LIN {X 0,Y 355.726,Z 424.465,A -85,B 0,C 180,E1 -13380.407,E2 -13380.407} C_VEL
LIN {X 0,Y 354.984,Z 431.448,A -85,B 0,C 180,E1 -13384.185,E2 -13384.185} C_VEL
LIN {X 0,Y 354.319,Z 439.711,A -85,B 0,C 180,E1 -13388.41,E2 -13388.41} C_VEL
LIN {X 0,Y 357.709,Z 454.995,A -85,B 0,C 180,E1 -13389.372,E2 -13389.372} C_VEL
LIN {X 0,Y 359.439,Z 467.166,A -85,B 0,C 180,E1 -13390.263,E2 -13390.263} C_VEL
LIN {X 0,Y 360.148,Z 480.167,A -85,B 0,C 180,E1 -13391.37,E2 -13391.37} C_VEL
LIN {X 0,Y 359.701,Z 487.628,A -85,B 0,C 180,E1 -13392.082,E2 -13392.082} C_VEL
LIN {X 0,Y 358.234,Z 498.948,A -85,B 0,C 180,E1 -13393.331,E2 -13393.331} C_VEL
LIN {X 0,Y 356.998,Z 508.224,A -85,B 0,C 180,E1 -13394.593,E2 -13394.593} C_VEL
LIN {X 0,Y 356.085,Z 516.778,A -85,B 0,C 180,E1 -13396.013,E2 -13396.013} C_VEL
LIN {X 0,Y 355.032,Z 525.202,A -85,B 0,C 180,E1 -13397.718,E2 -13397.718} C_VEL
LIN {X 0,Y 354.24,Z 532.058,A -85,B 0,C 180,E1 -13399.43,E2 -13399.43} C_VEL
LIN {X 0,Y 353.672,Z 538.425,A -85,B 0,C 180,E1 -13401.433,E2 -13401.433} C_VEL
LIN {X 0,Y 353.414,Z 542.602,A -85,B 0,C 180,E1 -13403.152,E2 -13403.152} C_VEL
LIN {X 0,Y 353.311,Z 544.771,A -85,B 0,C 180,E1 -13404.296,E2 -13404.296} C_VEL
LIN {X 0,Y 353.316,Z 546.521,A -85,B 0,C 180,E1 -13405.441,E2 -13405.441} C_VEL
LIN {X 0,Y 353.284,Z 547.858,A -85,B 0,C 180,E1 -13406.583,E2 -13406.583} C_VEL
LIN {X 0,Y 353.35,Z 548.753,A -85,B 0,C 180,E1 -13407.724,E2 -13407.724} C_VEL
LIN {X 0,Y 353.463,Z 549.226,A -85,B 0,C 180,E1 -13408.865,E2 -13408.865} C_VEL
LIN {X 0,Y 353.456,Z 549.291,A -85,B 0,C 180,E1 -13410.004,E2 -13410.004} C_VEL
LIN {X 0,Y 353.47,Z 548.959,A -85,B 0,C 180,E1 -13411.143,E2 -13411.143} C_VEL
LIN {X 0,Y 353.41,Z 548.175,A -85,B 0,C 180,E1 -13412.284,E2 -13412.284} C_VEL
LIN {X 0,Y 353.313,Z 546.954,A -85,B 0,C 180,E1 -13413.425,E2 -13413.425} C_VEL
LIN {X 0,Y 353.368,Z 544.327,A -85,B 0,C 180,E1 -13415.139,E2 -13415.139} C_VEL
LIN {X 0,Y 353.432,Z 540.637,A -85,B 0,C 180,E1 -13416.856,E2 -13416.856} C_VEL
LIN {X 0,Y 353.674,Z 535.798,A -85,B 0,C 180,E1 -13418.575,E2 -13418.575} C_VEL
LIN {X 0,Y 354.06,Z 529.666,A -85,B 0,C 180,E1 -13420.295,E2 -13420.295} C_VEL
LIN {X 0,Y 354.749,Z 522.044,A -85,B 0,C 180,E1 -13422.01,E2 -13422.01} C_VEL
LIN {X 0,Y 355.442,Z 514.243,A -85,B 0,C 180,E1 -13423.438,E2 -13423.438} C_VEL
LIN {X 0,Y 356.383,Z 503.675,A -85,B 0,C 180,E1 -13425.004,E2 -13425.004} C_VEL
LIN {X 0,Y 357.344,Z 493,A -85,B 0,C 180,E1 -13426.279,E2 -13426.279} C_VEL
LIN {X 0,Y 358.499,Z 481.057,A -85,B 0,C 180,E1 -13427.399,E2 -13427.399} C_VEL
LIN {X 0,Y 357.508,Z 469.159,A -85,B 0,C 180,E1 -13428.336,E2 -13428.336} C_VEL
LIN {X 0,Y 355.884,Z 455.898,A -85,B 0,C 180,E1 -13429.157,E2 -13429.157} C_VEL
LIN {X 0,Y 354,Z 442.82,A -85,B 0,C 180,E1 -13429.766,E2 -13429.766} C_VEL
LIN {X 0,Y 354.506,Z 435.528,A -85,B 0,C 180,E1 -13433.363,E2 -13433.363} C_VEL
LIN {X 0,Y 355.125,Z 428.123,A -85,B 0,C 180,E1 -13437.08,E2 -13437.08} C_VEL
LIN {X 0,Y 355.948,Z 420.705,A -85,B 0,C 180,E1 -13440.891,E2 -13440.891} C_VEL
LIN {X 0,Y 356.669,Z 414.53,A -85,B 0,C 180,E1 -13444.147,E2 -13444.147} C_VEL
LIN {X 0,Y 357.086,Z 410.748,A -85,B 0,C 180,E1 -13446.2,E2 -13446.2} C_VEL
LIN {X 0,Y 356.797,Z 407.568,A -85,B 0,C 180,E1 -13448.009,E2 -13448.009} C_VEL
LIN {X 0,Y 355.865,Z 401.962,A -85,B 0,C 180,E1 -13451.368,E2 -13451.368} C_VEL
LIN {X 0,Y 354.819,Z 396.286,A -85,B 0,C 180,E1 -13454.988,E2 -13454.988} C_VEL
LIN {X 0,Y 354.786,Z 396.293,A -85,B 0,C 180,E1 -13458.833,E2 -13458.833} C_VEL
LIN {X 0,Y 354.814,Z 396.285,A -85,B 0,C 180,E1 -13462.406,E2 -13462.406} C_VEL
LIN {X 0,Y 354.823,Z 396.288,A -85,B 0,C 180,E1 -13464.941,E2 -13464.941} C_VEL
LIN {X 0,Y 354.808,Z 396.287,A -85,B 0,C 180,E1 -13468.406,E2 -13468.406} C_VEL
LIN {X 0,Y 354.817,Z 396.287,A -85,B 0,C 180,E1 -13471.615,E2 -13471.615} C_VEL
LIN {X 0,Y 354.85,Z 396.282,A -85,B 0,C 180,E1 -13475.657,E2 -13475.657} C_VEL
LIN {X 0,Y 354.841,Z 396.287,A -85,B 0,C 180,E1 -13479.113,E2 -13479.113} C_VEL
LIN {X 0,Y 354.895,Z 396.278,A -85,B 0,C 180,E1 -13482.719,E2 -13482.719} C_VEL
LIN {X 0,Y 354.966,Z 396.266,A -85,B 0,C 180,E1 -13486.255,E2 -13486.255} C_VEL
LIN {X 0,Y 354.969,Z 396.266,A -85,B 0,C 180,E1 -13489.735,E2 -13489.735} C_VEL
LIN {X 0,Y 355.12,Z 396.251,A -85,B 0,C 180,E1 -13493.179,E2 -13493.179} C_VEL
LIN {X 0,Y 355.254,Z 396.231,A -85,B 0,C 180,E1 -13497.731,E2 -13497.731} C_VEL
LIN {X 0,Y 355.345,Z 396.219,A -85,B 0,C 180,E1 -13499.999,E2 -13499.999} C_VEL
LIN {X 0,Y 355.246,Z 396.233,A -85,B 0,C 180,E1 -13502.267,E2 -13502.267} C_VEL
LIN {X 0,Y 355.1,Z 396.255,A -85,B 0,C 180,E1 -13506.819,E2 -13506.819} C_VEL
LIN {X 0,Y 354.967,Z 396.268,A -85,B 0,C 180,E1 -13510.263,E2 -13510.263} C_VEL
LIN {X 0,Y 354.955,Z 396.268,A -85,B 0,C 180,E1 -13514.017,E2 -13514.017} C_VEL
LIN {X 0,Y 354.902,Z 396.275,A -85,B 0,C 180,E1 -13518.09,E2 -13518.09} C_VEL
LIN {X 0,Y 354.826,Z 396.285,A -85,B 0,C 180,E1 -13522.105,E2 -13522.105} C_VEL
LIN {X 0,Y 354.908,Z 396.274,A -85,B 0,C 180,E1 -13525.825,E2 -13525.825} C_VEL
LIN {X 0,Y 354.815,Z 396.285,A -85,B 0,C 180,E1 -13529.681,E2 -13529.681} C_VEL
LIN {X 0,Y 354.824,Z 396.284,A -85,B 0,C 180,E1 -13533.681,E2 -13533.681} C_VEL
LIN {X 0,Y 354.805,Z 396.291,A -85,B 0,C 180,E1 -13536.457,E2 -13536.457} C_VEL
LIN {X 0,Y 354.807,Z 396.286,A -85,B 0,C 180,E1 -13539.416,E2 -13539.416} C_VEL
LIN {X 0,Y 354.794,Z 396.291,A -85,B 0,C 180,E1 -13542.864,E2 -13542.864} C_VEL
LIN {X 0,Y 354.772,Z 396.293,A -85,B 0,C 180,E1 -13546.1,E2 -13546.1} C_VEL
LIN {X 0,Y 354.79,Z 396.289,A -85,B 0,C 180,E1 -13549.175,E2 -13549.175} C_VEL
LIN {X 0,Y 354.81,Z 396.291,A -85,B 0,C 180,E1 -13552.4,E2 -13552.4} C_VEL
LIN {X 0,Y 354.816,Z 396.287,A -85,B 0,C 180,E1 -13554.937,E2 -13554.937} C_VEL
LIN {X 0,Y 354.797,Z 396.292,A -85,B 0,C 180,E1 -13558.402,E2 -13558.402} C_VEL
LIN {X 0,Y 354.849,Z 396.281,A -85,B 0,C 180,E1 -13561.615,E2 -13561.615} C_VEL
LIN {X 0,Y 354.901,Z 396.279,A -85,B 0,C 180,E1 -13564.169,E2 -13564.169} C_VEL
LIN {X 0,Y 354.836,Z 396.285,A -85,B 0,C 180,E1 -13567.89,E2 -13567.89} C_VEL
LIN {X 0,Y 354.922,Z 396.274,A -85,B 0,C 180,E1 -13571.888,E2 -13571.888} C_VEL
LIN {X 0,Y 354.941,Z 396.273,A -85,B 0,C 180,E1 -13575.977,E2 -13575.977} C_VEL
LIN {X 0,Y 354.975,Z 396.267,A -85,B 0,C 180,E1 -13579.732,E2 -13579.732} C_VEL
LIN {X 0,Y 355.12,Z 396.247,A -85,B 0,C 180,E1 -13583.176,E2 -13583.176} C_VEL
LIN {X 0,Y 355.237,Z 396.235,A -85,B 0,C 180,E1 -13587.728,E2 -13587.728} C_VEL
LIN {X 0,Y 355.388,Z 396.218,A -85,B 0,C 180,E1 -13589.996,E2 -13589.996} C_VEL
LIN {X 0,Y 355.237,Z 396.238,A -85,B 0,C 180,E1 -13592.263,E2 -13592.263} C_VEL
LIN {X 0,Y 355.128,Z 396.247,A -85,B 0,C 180,E1 -13596.815,E2 -13596.815} C_VEL
LIN {X 0,Y 355.005,Z 396.262,A -85,B 0,C 180,E1 -13599.108,E2 -13599.108} C_VEL
LIN {X 0,Y 354.913,Z 396.275,A -85,B 0,C 180,E1 -13602.576,E2 -13602.576} C_VEL
LIN {X 0,Y 354.877,Z 396.283,A -85,B 0,C 180,E1 -13606.092,E2 -13606.092} C_VEL
LIN {X 0,Y 354.89,Z 396.278,A -85,B 0,C 180,E1 -13608.468,E2 -13608.468} C_VEL
LIN {X 0,Y 354.816,Z 396.29,A -85,B 0,C 180,E1 -13612.102,E2 -13612.102} C_VEL
LIN {X 0,Y 354.828,Z 396.284,A -85,B 0,C 180,E1 -13614.573,E2 -13614.573} C_VEL
LIN {X 0,Y 354.671,Z 396.303,A -85,B 0,C 180,E1 -13617.108,E2 -13617.108} C_VEL
LIN {X 0,Y 354.374,Z 396.345,A -85,B 0,C 180,E1 -13619.717,E2 -13619.717} C_VEL
LIN {X 0,Y 354.027,Z 396.387,A -85,B 0,C 180,E1 -13622.405,E2 -13622.405} C_VEL
LIN {X 0,Y 353.895,Z 396.822,A -85,B 0,C 180,E1 -13623.777,E2 -13623.777} C_VEL
LIN {X 0,Y 353.774,Z 400.146,A -85,B 0,C 180,E1 -13627.382,E2 -13627.382} C_VEL
LIN {X 0,Y 353.684,Z 403.57,A -85,B 0,C 180,E1 -13630.969,E2 -13630.969} C_VEL
LIN {X 0,Y 353.68,Z 404.977,A -85,B 0,C 180,E1 -13632.398,E2 -13632.398} C_VEL
LIN {X 0,Y 356.886,Z 418.397,A -85,B 0,C 180,E1 -13633.129,E2 -13633.129} C_VEL
LIN {X 0,Y 359.642,Z 431.249,A -85,B 0,C 180,E1 -13634.039,E2 -13634.039} C_VEL
LIN {X 0,Y 359.648,Z 436.037,A -85,B 0,C 180,E1 -13634.399,E2 -13634.399} C_VEL
LIN {X 0,Y 358.833,Z 447.243,A -85,B 0,C 180,E1 -13635.363,E2 -13635.363} C_VEL
LIN {X 0,Y 357.756,Z 458.778,A -85,B 0,C 180,E1 -13636.615,E2 -13636.615} C_VEL
LIN {X 0,Y 357.607,Z 460.555,A -85,B 0,C 180,E1 -13636.835,E2 -13636.835} C_VEL
LIN {X 0,Y 356.539,Z 465.133,A -85,B 0,C 180,E1 -13637.412,E2 -13637.412} C_VEL
LIN {X 0,Y 353.076,Z 472.268,A -85,B 0,C 180,E1 -13638.376,E2 -13638.376} C_VEL
LIN {X 0,Y 349.606,Z 478.873,A -85,B 0,C 180,E1 -13639.445,E2 -13639.445} C_VEL
LIN {X 0,Y 348.543,Z 482.621,A -85,B 0,C 180,E1 -13640.176,E2 -13640.176} C_VEL
LIN {X 0,Y 347.827,Z 490.364,A -85,B 0,C 180,E1 -13641.991,E2 -13641.991} C_VEL
LIN {X 0,Y 347.238,Z 496.207,A -85,B 0,C 180,E1 -13643.702,E2 -13643.702} C_VEL
LIN {X 0,Y 346.846,Z 500.886,A -85,B 0,C 180,E1 -13645.436,E2 -13645.436} C_VEL
LIN {X 0,Y 346.507,Z 504.996,A -85,B 0,C 180,E1 -13647.489,E2 -13647.489} C_VEL
LIN {X 0,Y 346.224,Z 507.705,A -85,B 0,C 180,E1 -13649.506,E2 -13649.506} C_VEL
LIN {X 0,Y 346.209,Z 508.83,A -85,B 0,C 180,E1 -13650.845,E2 -13650.845} C_VEL
LIN {X 0,Y 346.169,Z 509.366,A -85,B 0,C 180,E1 -13652.165,E2 -13652.165} C_VEL
LIN {X 0,Y 346.207,Z 509.422,A -85,B 0,C 180,E1 -13653.476,E2 -13653.476} C_VEL
LIN {X 0,Y 346.334,Z 508.95,A -85,B 0,C 180,E1 -13654.778,E2 -13654.778} C_VEL
LIN {X 0,Y 346.526,Z 507.981,A -85,B 0,C 180,E1 -13656.071,E2 -13656.071} C_VEL
LIN {X 0,Y 346.814,Z 506.542,A -85,B 0,C 180,E1 -13657.356,E2 -13657.356} C_VEL
LIN {X 0,Y 347.305,Z 503.406,A -85,B 0,C 180,E1 -13659.261,E2 -13659.261} C_VEL
LIN {X 0,Y 347.906,Z 499.097,A -85,B 0,C 180,E1 -13661.144,E2 -13661.144} C_VEL
LIN {X 0,Y 348.766,Z 493.475,A -85,B 0,C 180,E1 -13663.012,E2 -13663.012} C_VEL
LIN {X 0,Y 349.903,Z 486.366,A -85,B 0,C 180,E1 -13664.865,E2 -13664.865} C_VEL
LIN {X 0,Y 351.209,Z 477.432,A -85,B 0,C 180,E1 -13666.697,E2 -13666.697} C_VEL
LIN {X 0,Y 352.565,Z 467.814,A -85,B 0,C 180,E1 -13668.283,E2 -13668.283} C_VEL
LIN {X 0,Y 353.916,Z 458.132,A -85,B 0,C 180,E1 -13669.561,E2 -13669.561} C_VEL
LIN {X 0,Y 355.189,Z 447.027,A -85,B 0,C 180,E1 -13670.75,E2 -13670.75} C_VEL
LIN {X 0,Y 356.058,Z 438.589,A -85,B 0,C 180,E1 -13671.487,E2 -13671.487} C_VEL
LIN {X 0,Y 354.629,Z 430.955,A -85,B 0,C 180,E1 -13672.218,E2 -13672.218} C_VEL
LIN {X 0,Y 351.014,Z 418.776,A -85,B 0,C 180,E1 -13673.318,E2 -13673.318} C_VEL
LIN {X 0,Y 347.558,Z 409.355,A -85,B 0,C 180,E1 -13674.089,E2 -13674.089} C_VEL
LIN {X 0,Y 347.468,Z 408.819,A -85,B 0,C 180,E1 -13674.124,E2 -13674.124} C_VEL
LIN {X 0,Y 347.648,Z 405.401,A -85,B 0,C 180,E1 -13678.843,E2 -13678.843} C_VEL
LIN {X 0,Y 348.104,Z 403.772,A -85,B 0,C 180,E1 -13681.158,E2 -13681.158} C_VEL
LIN {X 0,Y 348.199,Z 400.872,A -85,B 0,C 180,E1 -13685.793,E2 -13685.793} C_VEL
LIN {X 0,Y 348.303,Z 399.27,A -85,B 0,C 180,E1 -13688.656,E2 -13688.656} C_VEL
LIN {X 0,Y 347.865,Z 397.31,A -85,B 0,C 180,E1 -13692.841,E2 -13692.841} C_VEL
LIN {X 0,Y 347.839,Z 397.157,A -85,B 0,C 180,E1 -13695.229,E2 -13695.229} C_VEL
LIN {X 0,Y 347.833,Z 397.16,A -85,B 0,C 180,E1 -13698.862,E2 -13698.862} C_VEL
LIN {X 0,Y 347.781,Z 397.163,A -85,B 0,C 180,E1 -13702.58,E2 -13702.58} C_VEL
LIN {X 0,Y 347.792,Z 397.164,A -85,B 0,C 180,E1 -13705.111,E2 -13705.111} C_VEL
LIN {X 0,Y 347.783,Z 397.162,A -85,B 0,C 180,E1 -13707.697,E2 -13707.697} C_VEL
LIN {X 0,Y 347.736,Z 397.171,A -85,B 0,C 180,E1 -13710.35,E2 -13710.35} C_VEL
LIN {X 0,Y 347.718,Z 397.171,A -85,B 0,C 180,E1 -13714.468,E2 -13714.468} C_VEL
LIN {X 0,Y 347.746,Z 397.169,A -85,B 0,C 180,E1 -13716.069,E2 -13716.069} C_VEL
LIN {X 0,Y 348.261,Z 399.777,A -85,B 0,C 180,E1 -13720.224,E2 -13720.224} C_VEL
LIN {X 0,Y 348.756,Z 402.481,A -85,B 0,C 180,E1 -13723.501,E2 -13723.501} C_VEL
LIN {X 0,Y 349.311,Z 405.852,A -85,B 0,C 180,E1 -13726.845,E2 -13726.845} C_VEL
LIN {X 0,Y 349.963,Z 409.541,A -85,B 0,C 180,E1 -13730.019,E2 -13730.019} C_VEL
LIN {X 0,Y 350.447,Z 413.541,A -85,B 0,C 180,E1 -13733.02,E2 -13733.02} C_VEL
LIN {X 0,Y 350.372,Z 415.65,A -85,B 0,C 180,E1 -13734.436,E2 -13734.436} C_VEL
LIN {X 0,Y 349.443,Z 420.778,A -85,B 0,C 180,E1 -13737.642,E2 -13737.642} C_VEL
LIN {X 0,Y 348.397,Z 427.812,A -85,B 0,C 180,E1 -13741.708,E2 -13741.708} C_VEL
LIN {X 0,Y 347.786,Z 433.661,A -85,B 0,C 180,E1 -13744.895,E2 -13744.895} C_VEL
LIN {X 0,Y 347.336,Z 439.222,A -85,B 0,C 180,E1 -13747.806,E2 -13747.806} C_VEL
LIN {X 0,Y 350.654,Z 453.448,A -85,B 0,C 180,E1 -13748.749,E2 -13748.749} C_VEL
LIN {X 0,Y 352.665,Z 466.488,A -85,B 0,C 180,E1 -13749.735,E2 -13749.735} C_VEL
LIN {X 0,Y 353.413,Z 479.258,A -85,B 0,C 180,E1 -13750.85,E2 -13750.85} C_VEL
LIN {X 0,Y 353.155,Z 486.716,A -85,B 0,C 180,E1 -13751.589,E2 -13751.589} C_VEL
LIN {X 0,Y 351.618,Z 498.048,A -85,B 0,C 180,E1 -13752.858,E2 -13752.858} C_VEL
LIN {X 0,Y 350.161,Z 508.316,A -85,B 0,C 180,E1 -13754.284,E2 -13754.284} C_VEL
LIN {X 0,Y 349.163,Z 516.792,A -85,B 0,C 180,E1 -13755.735,E2 -13755.735} C_VEL
LIN {X 0,Y 348.076,Z 525.127,A -85,B 0,C 180,E1 -13757.469,E2 -13757.469} C_VEL
LIN {X 0,Y 347.205,Z 531.924,A -85,B 0,C 180,E1 -13759.213,E2 -13759.213} C_VEL
LIN {X 0,Y 346.63,Z 538.191,A -85,B 0,C 180,E1 -13761.258,E2 -13761.258} C_VEL
LIN {X 0,Y 346.339,Z 542.311,A -85,B 0,C 180,E1 -13763.011,E2 -13763.011} C_VEL
LIN {X 0,Y 346.23,Z 544.459,A -85,B 0,C 180,E1 -13764.179,E2 -13764.179} C_VEL
LIN {X 0,Y 346.228,Z 546.191,A -85,B 0,C 180,E1 -13765.347,E2 -13765.347} C_VEL
LIN {X 0,Y 346.204,Z 547.505,A -85,B 0,C 180,E1 -13766.513,E2 -13766.513} C_VEL
LIN {X 0,Y 346.252,Z 548.363,A -85,B 0,C 180,E1 -13767.678,E2 -13767.678} C_VEL
LIN {X 0,Y 346.379,Z 548.818,A -85,B 0,C 180,E1 -13768.842,E2 -13768.842} C_VEL
LIN {X 0,Y 346.393,Z 548.866,A -85,B 0,C 180,E1 -13770.004,E2 -13770.004} C_VEL
LIN {X 0,Y 346.406,Z 548.506,A -85,B 0,C 180,E1 -13771.167,E2 -13771.167} C_VEL
LIN {X 0,Y 346.314,Z 547.681,A -85,B 0,C 180,E1 -13772.33,E2 -13772.33} C_VEL
LIN {X 0,Y 346.235,Z 546.439,A -85,B 0,C 180,E1 -13773.495,E2 -13773.495} C_VEL
LIN {X 0,Y 346.291,Z 543.763,A -85,B 0,C 180,E1 -13775.244,E2 -13775.244} C_VEL
LIN {X 0,Y 346.376,Z 540.02,A -85,B 0,C 180,E1 -13776.997,E2 -13776.997} C_VEL
LIN {X 0,Y 346.621,Z 535.123,A -85,B 0,C 180,E1 -13778.751,E2 -13778.751} C_VEL
LIN {X 0,Y 346.997,Z 528.923,A -85,B 0,C 180,E1 -13780.507,E2 -13780.507} C_VEL
LIN {X 0,Y 347.743,Z 521.212,A -85,B 0,C 180,E1 -13782.256,E2 -13782.256} C_VEL
LIN {X 0,Y 348.699,Z 511.532,A -85,B 0,C 180,E1 -13784,E2 -13784} C_VEL
LIN {X 0,Y 349.491,Z 502.638,A -85,B 0,C 180,E1 -13785.307,E2 -13785.307} C_VEL
LIN {X 0,Y 350.474,Z 491.799,A -85,B 0,C 180,E1 -13786.608,E2 -13786.608} C_VEL
LIN {X 0,Y 351.5,Z 481.346,A -85,B 0,C 180,E1 -13787.606,E2 -13787.606} C_VEL
LIN {X 0,Y 350.414,Z 468.521,A -85,B 0,C 180,E1 -13788.645,E2 -13788.645} C_VEL
LIN {X 0,Y 348.819,Z 455.316,A -85,B 0,C 180,E1 -13789.478,E2 -13789.478} C_VEL
LIN {X 0,Y 346.964,Z 442.526,A -85,B 0,C 180,E1 -13790.068,E2 -13790.068} C_VEL
LIN {X 0,Y 347.512,Z 435.034,A -85,B 0,C 180,E1 -13793.862,E2 -13793.862} C_VEL
LIN {X 0,Y 348.162,Z 427.64,A -85,B 0,C 180,E1 -13797.667,E2 -13797.667} C_VEL
LIN {X 0,Y 349.036,Z 420.236,A -85,B 0,C 180,E1 -13801.573,E2 -13801.573} C_VEL
LIN {X 0,Y 349.733,Z 414.795,A -85,B 0,C 180,E1 -13804.521,E2 -13804.521} C_VEL
LIN {X 0,Y 350.042,Z 411.112,A -85,B 0,C 180,E1 -13806.571,E2 -13806.571} C_VEL
LIN {X 0,Y 349.46,Z 406.488,A -85,B 0,C 180,E1 -13809.313,E2 -13809.313} C_VEL
LIN {X 0,Y 348.52,Z 401.195,A -85,B 0,C 180,E1 -13812.605,E2 -13812.605} C_VEL
LIN {X 0,Y 347.783,Z 397.163,A -85,B 0,C 180,E1 -13815.257,E2 -13815.257} C_VEL
LIN {X 0,Y 347.756,Z 397.168,A -85,B 0,C 180,E1 -13818.4,E2 -13818.4} C_VEL
LIN {X 0,Y 347.77,Z 397.164,A -85,B 0,C 180,E1 -13822.679,E2 -13822.679} C_VEL
LIN {X 0,Y 347.764,Z 397.164,A -85,B 0,C 180,E1 -13825.957,E2 -13825.957} C_VEL
LIN {X 0,Y 347.754,Z 397.166,A -85,B 0,C 180,E1 -13829.652,E2 -13829.652} C_VEL
LIN {X 0,Y 347.765,Z 397.165,A -85,B 0,C 180,E1 -13833.601,E2 -13833.601} C_VEL
LIN {X 0,Y 347.785,Z 397.161,A -85,B 0,C 180,E1 -13836.161,E2 -13836.161} C_VEL
LIN {X 0,Y 347.801,Z 397.159,A -85,B 0,C 180,E1 -13839.908,E2 -13839.908} C_VEL
LIN {X 0,Y 347.847,Z 397.154,A -85,B 0,C 180,E1 -13843.568,E2 -13843.568} C_VEL
LIN {X 0,Y 347.904,Z 397.151,A -85,B 0,C 180,E1 -13847.16,E2 -13847.16} C_VEL
LIN {X 0,Y 347.95,Z 397.143,A -85,B 0,C 180,E1 -13850.7,E2 -13850.7} C_VEL
LIN {X 0,Y 348.087,Z 397.128,A -85,B 0,C 180,E1 -13853.041,E2 -13853.041} C_VEL
LIN {X 0,Y 348.217,Z 397.107,A -85,B 0,C 180,E1 -13857.686,E2 -13857.686} C_VEL
LIN {X 0,Y 348.297,Z 397.097,A -85,B 0,C 180,E1 -13859.999,E2 -13859.999} C_VEL
LIN {X 0,Y 348.207,Z 397.109,A -85,B 0,C 180,E1 -13862.312,E2 -13862.312} C_VEL
LIN {X 0,Y 348.067,Z 397.13,A -85,B 0,C 180,E1 -13866.957,E2 -13866.957} C_VEL
LIN {X 0,Y 347.907,Z 397.148,A -85,B 0,C 180,E1 -13870.474,E2 -13870.474} C_VEL
LIN {X 0,Y 347.912,Z 397.146,A -85,B 0,C 180,E1 -13874.148,E2 -13874.148} C_VEL
LIN {X 0,Y 347.841,Z 397.156,A -85,B 0,C 180,E1 -13878.257,E2 -13878.257} C_VEL
LIN {X 0,Y 347.779,Z 397.162,A -85,B 0,C 180,E1 -13881.624,E2 -13881.624} C_VEL
LIN {X 0,Y 347.821,Z 397.159,A -85,B 0,C 180,E1 -13885.106,E2 -13885.106} C_VEL
LIN {X 0,Y 347.812,Z 397.157,A -85,B 0,C 180,E1 -13887.692,E2 -13887.692} C_VEL
LIN {X 0,Y 347.754,Z 397.164,A -85,B 0,C 180,E1 -13891.697,E2 -13891.697} C_VEL
LIN {X 0,Y 347.753,Z 397.169,A -85,B 0,C 180,E1 -13894.461,E2 -13894.461} C_VEL
LIN {X 0,Y 347.772,Z 397.163,A -85,B 0,C 180,E1 -13897.984,E2 -13897.984} C_VEL
LIN {X 0,Y 347.757,Z 397.165,A -85,B 0,C 180,E1 -13901.828,E2 -13901.828} C_VEL
LIN {X 0,Y 347.711,Z 397.172,A -85,B 0,C 180,E1 -13905.024,E2 -13905.024} C_VEL
LIN {X 0,Y 347.754,Z 397.169,A -85,B 0,C 180,E1 -13908.395,E2 -13908.395} C_VEL
LIN {X 0,Y 347.777,Z 397.164,A -85,B 0,C 180,E1 -13912.009,E2 -13912.009} C_VEL
LIN {X 0,Y 347.749,Z 397.165,A -85,B 0,C 180,E1 -13915.533,E2 -13915.533} C_VEL
LIN {X 0,Y 347.749,Z 397.17,A -85,B 0,C 180,E1 -13918.297,E2 -13918.297} C_VEL
LIN {X 0,Y 347.781,Z 397.162,A -85,B 0,C 180,E1 -13920.984,E2 -13920.984} C_VEL
LIN {X 0,Y 347.833,Z 397.155,A -85,B 0,C 180,E1 -13923.604,E2 -13923.604} C_VEL
LIN {X 0,Y 347.79,Z 397.164,A -85,B 0,C 180,E1 -13926.158,E2 -13926.158} C_VEL
LIN {X 0,Y 347.813,Z 397.159,A -85,B 0,C 180,E1 -13929.906,E2 -13929.906} C_VEL
LIN {X 0,Y 347.866,Z 397.156,A -85,B 0,C 180,E1 -13932.355,E2 -13932.355} C_VEL
LIN {X 0,Y 347.896,Z 397.15,A -85,B 0,C 180,E1 -13935.967,E2 -13935.967} C_VEL
LIN {X 0,Y 347.926,Z 397.144,A -85,B 0,C 180,E1 -13939.522,E2 -13939.522} C_VEL
LIN {X 0,Y 348.086,Z 397.124,A -85,B 0,C 180,E1 -13943.038,E2 -13943.038} C_VEL
LIN {X 0,Y 348.199,Z 397.111,A -85,B 0,C 180,E1 -13947.682,E2 -13947.682} C_VEL
LIN {X 0,Y 348.337,Z 397.096,A -85,B 0,C 180,E1 -13949.996,E2 -13949.996} C_VEL
LIN {X 0,Y 348.2,Z 397.114,A -85,B 0,C 180,E1 -13952.309,E2 -13952.309} C_VEL
LIN {X 0,Y 348.096,Z 397.122,A -85,B 0,C 180,E1 -13956.953,E2 -13956.953} C_VEL
LIN {X 0,Y 347.958,Z 397.139,A -85,B 0,C 180,E1 -13959.294,E2 -13959.294} C_VEL
LIN {X 0,Y 347.881,Z 397.149,A -85,B 0,C 180,E1 -13962.835,E2 -13962.835} C_VEL
LIN {X 0,Y 347.826,Z 397.158,A -85,B 0,C 180,E1 -13966.427,E2 -13966.427} C_VEL
LIN {X 0,Y 347.839,Z 397.154,A -85,B 0,C 180,E1 -13968.856,E2 -13968.856} C_VEL
LIN {X 0,Y 347.755,Z 397.166,A -85,B 0,C 180,E1 -13972.575,E2 -13972.575} C_VEL
LIN {X 0,Y 347.74,Z 397.166,A -85,B 0,C 180,E1 -13975.108,E2 -13975.108} C_VEL
LIN {X 0,Y 347.558,Z 397.193,A -85,B 0,C 180,E1 -13977.71,E2 -13977.71} C_VEL
LIN {X 0,Y 347.222,Z 397.234,A -85,B 0,C 180,E1 -13980.393,E2 -13980.393} C_VEL
LIN {X 0,Y 346.874,Z 397.281,A -85,B 0,C 180,E1 -13983.158,E2 -13983.158} C_VEL
LIN {X 0,Y 346.783,Z 398.296,A -85,B 0,C 180,E1 -13984.567,E2 -13984.567} C_VEL
LIN {X 0,Y 346.709,Z 401.251,A -85,B 0,C 180,E1 -13987.765,E2 -13987.765} C_VEL
LIN {X 0,Y 346.62,Z 404.687,A -85,B 0,C 180,E1 -13991.394,E2 -13991.394} C_VEL
LIN {X 0,Y 346.611,Z 405.334,A -85,B 0,C 180,E1 -13992.065,E2 -13992.065} C_VEL
LIN {X 0,Y 349.954,Z 419.396,A -85,B 0,C 180,E1 -13992.86,E2 -13992.86} C_VEL
LIN {X 0,Y 352.739,Z 432.353,A -85,B 0,C 180,E1 -13993.813,E2 -13993.813} C_VEL
LIN {X 0,Y 352.805,Z 435.767,A -85,B 0,C 180,E1 -13994.081,E2 -13994.081} C_VEL
LIN {X 0,Y 351.977,Z 447.134,A -85,B 0,C 180,E1 -13995.064,E2 -13995.064} C_VEL
LIN {X 0,Y 350.848,Z 458.924,A -85,B 0,C 180,E1 -13996.36,E2 -13996.36} C_VEL
LIN {X 0,Y 349.959,Z 468.818,A -85,B 0,C 180,E1 -13997.715,E2 -13997.715} C_VEL
LIN {X 0,Y 349.131,Z 477.37,A -85,B 0,C 180,E1 -13999.141,E2 -13999.141} C_VEL
LIN {X 0,Y 348.543,Z 482.621,A -85,B 0,C 180,E1 -14000.176,E2 -14000.176} C_VEL
LIN {X 0,Y 347.5,Z 486.196,A -85,B 0,C 180,E1 -14000.937,E2 -14000.937} C_VEL
LIN {X 0,Y 344.134,Z 491.575,A -85,B 0,C 180,E1 -14002.201,E2 -14002.201} C_VEL
LIN {X 0,Y 340.868,Z 496.35,A -85,B 0,C 180,E1 -14003.551,E2 -14003.551} C_VEL
LIN {X 0,Y 339.996,Z 498.892,A -85,B 0,C 180,E1 -14004.433,E2 -14004.433} C_VEL
LIN {X 0,Y 339.684,Z 502.72,A -85,B 0,C 180,E1 -14006.041,E2 -14006.041} C_VEL
LIN {X 0,Y 339.297,Z 506.409,A -85,B 0,C 180,E1 -14008.119,E2 -14008.119} C_VEL
LIN {X 0,Y 339.093,Z 508.953,A -85,B 0,C 180,E1 -14010.503,E2 -14010.503} C_VEL
LIN {X 0,Y 339.102,Z 509.898,A -85,B 0,C 180,E1 -14012.875,E2 -14012.875} C_VEL
LIN {X 0,Y 339.175,Z 509.687,A -85,B 0,C 180,E1 -14014.207,E2 -14014.207} C_VEL
LIN {X 0,Y 339.387,Z 508.936,A -85,B 0,C 180,E1 -14015.65,E2 -14015.65} C_VEL
LIN {X 0,Y 339.604,Z 507.816,A -85,B 0,C 180,E1 -14016.848,E2 -14016.848} C_VEL
LIN {X 0,Y 340.017,Z 505.713,A -85,B 0,C 180,E1 -14018.438,E2 -14018.438} C_VEL
LIN {X 0,Y 340.495,Z 502.666,A -85,B 0,C 180,E1 -14020.09,E2 -14020.09} C_VEL
LIN {X 0,Y 341.243,Z 497.987,A -85,B 0,C 180,E1 -14022.006,E2 -14022.006} C_VEL
LIN {X 0,Y 342.236,Z 491.939,A -85,B 0,C 180,E1 -14023.906,E2 -14023.906} C_VEL
LIN {X 0,Y 343.496,Z 484.34,A -85,B 0,C 180,E1 -14025.788,E2 -14025.788} C_VEL
LIN {X 0,Y 344.889,Z 475.659,A -85,B 0,C 180,E1 -14027.504,E2 -14027.504} C_VEL
LIN {X 0,Y 346.26,Z 466.039,A -85,B 0,C 180,E1 -14029.032,E2 -14029.032} C_VEL
LIN {X 0,Y 347.793,Z 455.262,A -85,B 0,C 180,E1 -14030.404,E2 -14030.404} C_VEL
LIN {X 0,Y 349.182,Z 443.284,A -85,B 0,C 180,E1 -14031.61,E2 -14031.61} C_VEL
LIN {X 0,Y 349.567,Z 439.816,A -85,B 0,C 180,E1 -14031.911,E2 -14031.911} C_VEL
LIN {X 0,Y 347.536,Z 430.249,A -85,B 0,C 180,E1 -14032.886,E2 -14032.886} C_VEL
LIN {X 0,Y 343.843,Z 418.356,A -85,B 0,C 180,E1 -14033.994,E2 -14033.994} C_VEL
LIN {X 0,Y 340.492,Z 409.761,A -85,B 0,C 180,E1 -14034.746,E2 -14034.746} C_VEL
LIN {X 0,Y 340.429,Z 409.341,A -85,B 0,C 180,E1 -14034.819,E2 -14034.819} C_VEL
LIN {X 0,Y 340.876,Z 405.701,A -85,B 0,C 180,E1 -14040.001,E2 -14040.001} C_VEL
LIN {X 0,Y 341.101,Z 404.891,A -85,B 0,C 180,E1 -14041.182,E2 -14041.182} C_VEL
LIN {X 0,Y 341.211,Z 402.029,A -85,B 0,C 180,E1 -14045.912,E2 -14045.912} C_VEL
LIN {X 0,Y 341.298,Z 400.506,A -85,B 0,C 180,E1 -14048.771,E2 -14048.771} C_VEL
LIN {X 0,Y 340.988,Z 399.062,A -85,B 0,C 180,E1 -14051.895,E2 -14051.895} C_VEL
LIN {X 0,Y 340.83,Z 398.112,A -85,B 0,C 180,E1 -14054.327,E2 -14054.327} C_VEL
LIN {X 0,Y 340.809,Z 398.032,A -85,B 0,C 180,E1 -14058.471,E2 -14058.471} C_VEL
LIN {X 0,Y 340.75,Z 398.041,A -85,B 0,C 180,E1 -14061.871,E2 -14061.871} C_VEL
LIN {X 0,Y 340.748,Z 398.04,A -85,B 0,C 180,E1 -14065.667,E2 -14065.667} C_VEL
LIN {X 0,Y 340.713,Z 398.045,A -85,B 0,C 180,E1 -14068.323,E2 -14068.323} C_VEL
LIN {X 0,Y 340.676,Z 398.047,A -85,B 0,C 180,E1 -14071.048,E2 -14071.048} C_VEL
LIN {X 0,Y 340.697,Z 398.046,A -85,B 0,C 180,E1 -14074.409,E2 -14074.409} C_VEL
LIN {X 0,Y 341.034,Z 400.029,A -85,B 0,C 180,E1 -14078.189,E2 -14078.189} C_VEL
LIN {X 0,Y 341.472,Z 402.136,A -85,B 0,C 180,E1 -14081.195,E2 -14081.195} C_VEL
LIN {X 0,Y 341.954,Z 404.815,A -85,B 0,C 180,E1 -14084.331,E2 -14084.331} C_VEL
LIN {X 0,Y 342.518,Z 408.185,A -85,B 0,C 180,E1 -14087.619,E2 -14087.619} C_VEL
LIN {X 0,Y 343.182,Z 412.316,A -85,B 0,C 180,E1 -14091.097,E2 -14091.097} C_VEL
LIN {X 0,Y 343.466,Z 414.77,A -85,B 0,C 180,E1 -14092.942,E2 -14092.942} C_VEL
LIN {X 0,Y 343.208,Z 417.809,A -85,B 0,C 180,E1 -14095.021,E2 -14095.021} C_VEL
LIN {X 0,Y 342.163,Z 423.235,A -85,B 0,C 180,E1 -14098.421,E2 -14098.421} C_VEL
LIN {X 0,Y 341.238,Z 429.903,A -85,B 0,C 180,E1 -14102.328,E2 -14102.328} C_VEL
LIN {X 0,Y 340.494,Z 437.054,A -85,B 0,C 180,E1 -14106.272,E2 -14106.272} C_VEL
LIN {X 0,Y 340.345,Z 438.725,A -85,B 0,C 180,E1 -14107.17,E2 -14107.17} C_VEL
LIN {X 0,Y 343.796,Z 452.918,A -85,B 0,C 180,E1 -14108.148,E2 -14108.148} C_VEL
LIN {X 0,Y 345.789,Z 465.241,A -85,B 0,C 180,E1 -14109.126,E2 -14109.126} C_VEL
LIN {X 0,Y 346.636,Z 476.739,A -85,B 0,C 180,E1 -14110.152,E2 -14110.152} C_VEL
LIN {X 0,Y 346.625,Z 485.886,A -85,B 0,C 180,E1 -14111.075,E2 -14111.075} C_VEL
LIN {X 0,Y 345.011,Z 497.275,A -85,B 0,C 180,E1 -14112.367,E2 -14112.367} C_VEL
LIN {X 0,Y 343.624,Z 506.626,A -85,B 0,C 180,E1 -14113.672,E2 -14113.672} C_VEL
LIN {X 0,Y 342.358,Z 515.63,A -85,B 0,C 180,E1 -14115.204,E2 -14115.204} C_VEL
LIN {X 0,Y 341.289,Z 523.793,A -85,B 0,C 180,E1 -14116.913,E2 -14116.913} C_VEL
LIN {X 0,Y 340.286,Z 530.749,A -85,B 0,C 180,E1 -14118.69,E2 -14118.69} C_VEL
LIN {X 0,Y 339.713,Z 536.366,A -85,B 0,C 180,E1 -14120.478,E2 -14120.478} C_VEL
LIN {X 0,Y 339.367,Z 540.802,A -85,B 0,C 180,E1 -14122.269,E2 -14122.269} C_VEL
LIN {X 0,Y 339.171,Z 544.168,A -85,B 0,C 180,E1 -14124.058,E2 -14124.058} C_VEL
LIN {X 0,Y 339.125,Z 545.872,A -85,B 0,C 180,E1 -14125.249,E2 -14125.249} C_VEL
LIN {X 0,Y 339.126,Z 547.147,A -85,B 0,C 180,E1 -14126.44,E2 -14126.44} C_VEL
LIN {X 0,Y 339.297,Z 548.412,A -85,B 0,C 180,E1 -14128.818,E2 -14128.818} C_VEL
LIN {X 0,Y 339.332,Z 548.441,A -85,B 0,C 180,E1 -14130.004,E2 -14130.004} C_VEL
LIN {X 0,Y 339.324,Z 548.043,A -85,B 0,C 180,E1 -14131.191,E2 -14131.191} C_VEL
LIN {X 0,Y 339.219,Z 547.188,A -85,B 0,C 180,E1 -14132.379,E2 -14132.379} C_VEL
LIN {X 0,Y 339.158,Z 545.924,A -85,B 0,C 180,E1 -14133.568,E2 -14133.568} C_VEL
LIN {X 0,Y 339.197,Z 542.769,A -85,B 0,C 180,E1 -14135.593,E2 -14135.593} C_VEL
LIN {X 0,Y 339.373,Z 537.892,A -85,B 0,C 180,E1 -14137.74,E2 -14137.74} C_VEL
LIN {X 0,Y 339.773,Z 531.492,A -85,B 0,C 180,E1 -14139.829,E2 -14139.829} C_VEL
LIN {X 0,Y 340.308,Z 524.497,A -85,B 0,C 180,E1 -14141.62,E2 -14141.62} C_VEL
LIN {X 0,Y 341.176,Z 515.736,A -85,B 0,C 180,E1 -14143.404,E2 -14143.404} C_VEL
LIN {X 0,Y 341.9,Z 507.332,A -85,B 0,C 180,E1 -14144.805,E2 -14144.805} C_VEL
LIN {X 0,Y 343.04,Z 497.005,A -85,B 0,C 180,E1 -14146.213,E2 -14146.213} C_VEL
LIN {X 0,Y 344.108,Z 486.314,A -85,B 0,C 180,E1 -14147.383,E2 -14147.383} C_VEL
LIN {X 0,Y 344.493,Z 481.632,A -85,B 0,C 180,E1 -14147.823,E2 -14147.823} C_VEL
LIN {X 0,Y 343.476,Z 469.253,A -85,B 0,C 180,E1 -14148.864,E2 -14148.864} C_VEL
LIN {X 0,Y 341.86,Z 455.851,A -85,B 0,C 180,E1 -14149.754,E2 -14149.754} C_VEL
LIN {X 0,Y 339.933,Z 442.134,A -85,B 0,C 180,E1 -14150.423,E2 -14150.423} C_VEL
LIN {X 0,Y 340.506,Z 434.508,A -85,B 0,C 180,E1 -14154.385,E2 -14154.385} C_VEL
LIN {X 0,Y 341.232,Z 427.151,A -85,B 0,C 180,E1 -14158.279,E2 -14158.279} C_VEL
LIN {X 0,Y 342.146,Z 419.762,A -85,B 0,C 180,E1 -14162.284,E2 -14162.284} C_VEL
LIN {X 0,Y 343.012,Z 413.575,A -85,B 0,C 180,E1 -14165.732,E2 -14165.732} C_VEL
LIN {X 0,Y 342.79,Z 409.804,A -85,B 0,C 180,E1 -14167.961,E2 -14167.961} C_VEL
LIN {X 0,Y 341.944,Z 404.693,A -85,B 0,C 180,E1 -14171.129,E2 -14171.129} C_VEL
LIN {X 0,Y 341.003,Z 399.565,A -85,B 0,C 180,E1 -14174.49,E2 -14174.49} C_VEL
LIN {X 0,Y 340.739,Z 398.041,A -85,B 0,C 180,E1 -14175.578,E2 -14175.578} C_VEL
LIN {X 0,Y 340.686,Z 398.048,A -85,B 0,C 180,E1 -14178.689,E2 -14178.689} C_VEL
LIN {X 0,Y 340.734,Z 398.04,A -85,B 0,C 180,E1 -14181.772,E2 -14181.772} C_VEL
LIN {X 0,Y 340.738,Z 398.04,A -85,B 0,C 180,E1 -14185.597,E2 -14185.597} C_VEL
LIN {X 0,Y 340.709,Z 398.046,A -85,B 0,C 180,E1 -14188.955,E2 -14188.955} C_VEL
LIN {X 0,Y 340.736,Z 398.044,A -85,B 0,C 180,E1 -14193.013,E2 -14193.013} C_VEL
LIN {X 0,Y 340.757,Z 398.037,A -85,B 0,C 180,E1 -14195.637,E2 -14195.637} C_VEL
LIN {X 0,Y 340.736,Z 398.041,A -85,B 0,C 180,E1 -14199.473,E2 -14199.473} C_VEL
LIN {X 0,Y 340.808,Z 398.029,A -85,B 0,C 180,E1 -14201.981,E2 -14201.981} C_VEL
LIN {X 0,Y 340.869,Z 398.022,A -85,B 0,C 180,E1 -14205.716,E2 -14205.716} C_VEL
LIN {X 0,Y 340.862,Z 398.026,A -85,B 0,C 180,E1 -14209.305,E2 -14209.305} C_VEL
LIN {X 0,Y 341.056,Z 398.004,A -85,B 0,C 180,E1 -14212.897,E2 -14212.897} C_VEL
LIN {X 0,Y 341.179,Z 397.984,A -85,B 0,C 180,E1 -14217.638,E2 -14217.638} C_VEL
LIN {X 0,Y 341.249,Z 397.975,A -85,B 0,C 180,E1 -14219.999,E2 -14219.999} C_VEL
LIN {X 0,Y 341.145,Z 397.989,A -85,B 0,C 180,E1 -14222.36,E2 -14222.36} C_VEL
LIN {X 0,Y 341.003,Z 398.005,A -85,B 0,C 180,E1 -14226.556,E2 -14226.556} C_VEL
LIN {X 0,Y 340.894,Z 398.02,A -85,B 0,C 180,E1 -14229.492,E2 -14229.492} C_VEL
LIN {X 0,Y 340.856,Z 398.027,A -85,B 0,C 180,E1 -14233.108,E2 -14233.108} C_VEL
LIN {X 0,Y 340.787,Z 398.038,A -85,B 0,C 180,E1 -14236.78,E2 -14236.78} C_VEL
LIN {X 0,Y 340.739,Z 398.04,A -85,B 0,C 180,E1 -14239.268,E2 -14239.268} C_VEL
LIN {X 0,Y 340.732,Z 398.042,A -85,B 0,C 180,E1 -14243.071,E2 -14243.071} C_VEL
LIN {X 0,Y 340.782,Z 398.033,A -85,B 0,C 180,E1 -14245.662,E2 -14245.662} C_VEL
LIN {X 0,Y 340.729,Z 398.042,A -85,B 0,C 180,E1 -14248.319,E2 -14248.319} C_VEL
LIN {X 0,Y 340.704,Z 398.045,A -85,B 0,C 180,E1 -14251.043,E2 -14251.043} C_VEL
LIN {X 0,Y 340.726,Z 398.04,A -85,B 0,C 180,E1 -14255.276,E2 -14255.276} C_VEL
LIN {X 0,Y 340.703,Z 398.047,A -85,B 0,C 180,E1 -14258.38,E2 -14258.38} C_VEL
LIN {X 0,Y 340.705,Z 398.044,A -85,B 0,C 180,E1 -14262.042,E2 -14262.042} C_VEL
LIN {X 0,Y 340.658,Z 398.051,A -85,B 0,C 180,E1 -14266.224,E2 -14266.224} C_VEL
LIN {X 0,Y 340.691,Z 398.045,A -85,B 0,C 180,E1 -14269.75,E2 -14269.75} C_VEL
LIN {X 0,Y 340.709,Z 398.042,A -85,B 0,C 180,E1 -14273.255,E2 -14273.255} C_VEL
LIN {X 0,Y 340.697,Z 398.047,A -85,B 0,C 180,E1 -14276.15,E2 -14276.15} C_VEL
LIN {X 0,Y 340.745,Z 398.043,A -85,B 0,C 180,E1 -14280.326,E2 -14280.326} C_VEL
LIN {X 0,Y 340.806,Z 398.031,A -85,B 0,C 180,E1 -14283.016,E2 -14283.016} C_VEL
LIN {X 0,Y 340.758,Z 398.036,A -85,B 0,C 180,E1 -14285.635,E2 -14285.635} C_VEL
LIN {X 0,Y 340.745,Z 398.037,A -85,B 0,C 180,E1 -14289.47,E2 -14289.47} C_VEL
LIN {X 0,Y 340.857,Z 398.026,A -85,B 0,C 180,E1 -14291.98,E2 -14291.98} C_VEL
LIN {X 0,Y 340.868,Z 398.023,A -85,B 0,C 180,E1 -14295.701,E2 -14295.701} C_VEL
LIN {X 0,Y 340.868,Z 398.022,A -85,B 0,C 180,E1 -14299.302,E2 -14299.302} C_VEL
LIN {X 0,Y 341.054,Z 398,A -85,B 0,C 180,E1 -14302.894,E2 -14302.894} C_VEL
LIN {X 0,Y 341.161,Z 397.987,A -85,B 0,C 180,E1 -14307.634,E2 -14307.634} C_VEL
LIN {X 0,Y 341.287,Z 397.974,A -85,B 0,C 180,E1 -14309.996,E2 -14309.996} C_VEL
LIN {X 0,Y 341.161,Z 397.99,A -85,B 0,C 180,E1 -14312.357,E2 -14312.357} C_VEL
LIN {X 0,Y 341.065,Z 397.998,A -85,B 0,C 180,E1 -14317.097,E2 -14317.097} C_VEL
LIN {X 0,Y 340.863,Z 398.024,A -85,B 0,C 180,E1 -14320.689,E2 -14320.689} C_VEL
LIN {X 0,Y 340.849,Z 398.028,A -85,B 0,C 180,E1 -14324.32,E2 -14324.32} C_VEL
LIN {X 0,Y 340.822,Z 398.03,A -85,B 0,C 180,E1 -14328.463,E2 -14328.463} C_VEL
LIN {X 0,Y 340.736,Z 398.043,A -85,B 0,C 180,E1 -14331.853,E2 -14331.853} C_VEL
LIN {X 0,Y 340.713,Z 398.041,A -85,B 0,C 180,E1 -14334.827,E2 -14334.827} C_VEL
LIN {X 0,Y 340.541,Z 398.065,A -85,B 0,C 180,E1 -14337.452,E2 -14337.452} C_VEL
LIN {X 0,Y 340.097,Z 398.119,A -85,B 0,C 180,E1 -14341.099,E2 -14341.099} C_VEL
LIN {X 0,Y 339.763,Z 398.497,A -85,B 0,C 180,E1 -14343.945,E2 -14343.945} C_VEL
LIN {X 0,Y 339.627,Z 402.336,A -85,B 0,C 180,E1 -14348.157,E2 -14348.157} C_VEL
LIN {X 0,Y 339.544,Z 405.754,A -85,B 0,C 180,E1 -14351.739,E2 -14351.739} C_VEL
LIN {X 0,Y 342.671,Z 418.91,A -85,B 0,C 180,E1 -14352.483,E2 -14352.483} C_VEL
LIN {X 0,Y 345.335,Z 430.976,A -85,B 0,C 180,E1 -14353.374,E2 -14353.374} C_VEL
LIN {X 0,Y 346.008,Z 434.459,A -85,B 0,C 180,E1 -14353.67,E2 -14353.67} C_VEL
LIN {X 0,Y 345.139,Z 446.518,A -85,B 0,C 180,E1 -14354.707,E2 -14354.707} C_VEL
LIN {X 0,Y 344.191,Z 456.619,A -85,B 0,C 180,E1 -14355.792,E2 -14355.792} C_VEL
LIN {X 0,Y 343.124,Z 467.685,A -85,B 0,C 180,E1 -14357.277,E2 -14357.277} C_VEL
LIN {X 0,Y 342.179,Z 477.489,A -85,B 0,C 180,E1 -14358.912,E2 -14358.912} C_VEL
LIN {X 0,Y 341.229,Z 485.97,A -85,B 0,C 180,E1 -14360.673,E2 -14360.673} C_VEL
LIN {X 0,Y 340.521,Z 493,A -85,B 0,C 180,E1 -14362.495,E2 -14362.495} C_VEL
LIN {X 0,Y 339.996,Z 498.892,A -85,B 0,C 180,E1 -14364.433,E2 -14364.433} C_VEL
LIN {X 0,Y 339.128,Z 501.232,A -85,B 0,C 180,E1 -14365.337,E2 -14365.337} C_VEL
LIN {X 0,Y 335.937,Z 504.493,A -85,B 0,C 180,E1 -14366.834,E2 -14366.834} C_VEL
LIN {X 0,Y 332.813,Z 507.132,A -85,B 0,C 180,E1 -14368.394,E2 -14368.394} C_VEL
LIN {X 0,Y 332.069,Z 508.313,A -85,B 0,C 180,E1 -14369.385,E2 -14369.385} C_VEL
LIN {X 0,Y 332.018,Z 509.593,A -85,B 0,C 180,E1 -14370.867,E2 -14370.867} C_VEL
LIN {X 0,Y 332.005,Z 510.294,A -85,B 0,C 180,E1 -14372.743,E2 -14372.743} C_VEL
LIN {X 0,Y 332.185,Z 509.885,A -85,B 0,C 180,E1 -14374.969,E2 -14374.969} C_VEL
LIN {X 0,Y 332.417,Z 508.951,A -85,B 0,C 180,E1 -14376.317,E2 -14376.317} C_VEL
LIN {X 0,Y 332.893,Z 506.747,A -85,B 0,C 180,E1 -14378.251,E2 -14378.251} C_VEL
LIN {X 0,Y 333.512,Z 503.239,A -85,B 0,C 180,E1 -14380.297,E2 -14380.297} C_VEL
LIN {X 0,Y 334.299,Z 498.635,A -85,B 0,C 180,E1 -14382.253,E2 -14382.253} C_VEL
LIN {X 0,Y 335.364,Z 492.646,A -85,B 0,C 180,E1 -14384.192,E2 -14384.192} C_VEL
LIN {X 0,Y 336.703,Z 485.09,A -85,B 0,C 180,E1 -14386.112,E2 -14386.112} C_VEL
LIN {X 0,Y 338.033,Z 477.318,A -85,B 0,C 180,E1 -14387.705,E2 -14387.705} C_VEL
LIN {X 0,Y 339.449,Z 468.045,A -85,B 0,C 180,E1 -14389.262,E2 -14389.262} C_VEL
LIN {X 0,Y 341.105,Z 457.334,A -85,B 0,C 180,E1 -14390.695,E2 -14390.695} C_VEL
LIN {X 0,Y 342.532,Z 446.256,A -85,B 0,C 180,E1 -14391.892,E2 -14391.892} C_VEL
LIN {X 0,Y 343.079,Z 441.252,A -85,B 0,C 180,E1 -14392.349,E2 -14392.349} C_VEL
LIN {X 0,Y 340.562,Z 429.97,A -85,B 0,C 180,E1 -14393.543,E2 -14393.543} C_VEL
LIN {X 0,Y 336.47,Z 417.67,A -85,B 0,C 180,E1 -14394.758,E2 -14394.758} C_VEL
LIN {X 0,Y 333.537,Z 410.522,A -85,B 0,C 180,E1 -14395.431,E2 -14395.431} C_VEL
LIN {X 0,Y 333.416,Z 409.898,A -85,B 0,C 180,E1 -14395.505,E2 -14395.505} C_VEL
LIN {X 0,Y 333.853,Z 406.828,A -85,B 0,C 180,E1 -14400.001,E2 -14400.001} C_VEL
LIN {X 0,Y 334.119,Z 406.043,A -85,B 0,C 180,E1 -14401.206,E2 -14401.206} C_VEL
LIN {X 0,Y 334.225,Z 403.198,A -85,B 0,C 180,E1 -14406.036,E2 -14406.036} C_VEL
LIN {X 0,Y 334.292,Z 401.731,A -85,B 0,C 180,E1 -14408.887,E2 -14408.887} C_VEL
LIN {X 0,Y 333.988,Z 400.316,A -85,B 0,C 180,E1 -14412.148,E2 -14412.148} C_VEL
LIN {X 0,Y 333.851,Z 399.41,A -85,B 0,C 180,E1 -14414.633,E2 -14414.633} C_VEL
LIN {X 0,Y 333.726,Z 398.915,A -85,B 0,C 180,E1 -14417.148,E2 -14417.148} C_VEL
LIN {X 0,Y 333.728,Z 398.917,A -85,B 0,C 180,E1 -14419.692,E2 -14419.692} C_VEL
LIN {X 0,Y 333.688,Z 398.921,A -85,B 0,C 180,E1 -14423.59,E2 -14423.59} C_VEL
LIN {X 0,Y 333.709,Z 398.916,A -85,B 0,C 180,E1 -14426.25,E2 -14426.25} C_VEL
LIN {X 0,Y 333.683,Z 398.919,A -85,B 0,C 180,E1 -14428.976,E2 -14428.976} C_VEL
LIN {X 0,Y 333.641,Z 398.99,A -85,B 0,C 180,E1 -14432.597,E2 -14432.597} C_VEL
LIN {X 0,Y 333.912,Z 400.501,A -85,B 0,C 180,E1 -14436.111,E2 -14436.111} C_VEL
LIN {X 0,Y 334.259,Z 402.268,A -85,B 0,C 180,E1 -14439.108,E2 -14439.108} C_VEL
LIN {X 0,Y 334.797,Z 404.955,A -85,B 0,C 180,E1 -14442.726,E2 -14442.726} C_VEL
LIN {X 0,Y 335.329,Z 408.235,A -85,B 0,C 180,E1 -14446.248,E2 -14446.248} C_VEL
LIN {X 0,Y 335.946,Z 411.878,A -85,B 0,C 180,E1 -14449.577,E2 -14449.577} C_VEL
LIN {X 0,Y 336.47,Z 415.813,A -85,B 0,C 180,E1 -14452.725,E2 -14452.725} C_VEL
LIN {X 0,Y 336.304,Z 418.413,A -85,B 0,C 180,E1 -14454.59,E2 -14454.59} C_VEL
LIN {X 0,Y 335.344,Z 423.205,A -85,B 0,C 180,E1 -14457.702,E2 -14457.702} C_VEL
LIN {X 0,Y 334.47,Z 428.784,A -85,B 0,C 180,E1 -14461.106,E2 -14461.106} C_VEL
LIN {X 0,Y 333.659,Z 435.414,A -85,B 0,C 180,E1 -14464.923,E2 -14464.923} C_VEL
LIN {X 0,Y 333.409,Z 438.221,A -85,B 0,C 180,E1 -14466.484,E2 -14466.484} C_VEL
LIN {X 0,Y 334.233,Z 441.524,A -85,B 0,C 180,E1 -14466.701,E2 -14466.701} C_VEL
LIN {X 0,Y 337.305,Z 454.09,A -85,B 0,C 180,E1 -14467.656,E2 -14467.656} C_VEL
LIN {X 0,Y 339.105,Z 465.311,A -85,B 0,C 180,E1 -14468.589,E2 -14468.589} C_VEL
LIN {X 0,Y 339.953,Z 476.038,A -85,B 0,C 180,E1 -14469.587,E2 -14469.587} C_VEL
LIN {X 0,Y 339.94,Z 486.468,A -85,B 0,C 180,E1 -14470.689,E2 -14470.689} C_VEL
LIN {X 0,Y 338.272,Z 497.657,A -85,B 0,C 180,E1 -14472.003,E2 -14472.003} C_VEL
LIN {X 0,Y 336.818,Z 506.871,A -85,B 0,C 180,E1 -14473.332,E2 -14473.332} C_VEL
LIN {X 0,Y 335.433,Z 515.975,A -85,B 0,C 180,E1 -14474.943,E2 -14474.943} C_VEL
LIN {X 0,Y 334.367,Z 523.796,A -85,B 0,C 180,E1 -14476.637,E2 -14476.637} C_VEL
LIN {X 0,Y 333.294,Z 530.648,A -85,B 0,C 180,E1 -14478.449,E2 -14478.449} C_VEL
LIN {X 0,Y 332.692,Z 536.181,A -85,B 0,C 180,E1 -14480.275,E2 -14480.275} C_VEL
LIN {X 0,Y 332.302,Z 540.566,A -85,B 0,C 180,E1 -14482.103,E2 -14482.103} C_VEL
LIN {X 0,Y 332.074,Z 544.164,A -85,B 0,C 180,E1 -14484.108,E2 -14484.108} C_VEL
LIN {X 0,Y 332.049,Z 546.788,A -85,B 0,C 180,E1 -14486.364,E2 -14486.364} C_VEL
LIN {X 0,Y 332.201,Z 548.003,A -85,B 0,C 180,E1 -14488.792,E2 -14488.792} C_VEL
LIN {X 0,Y 332.272,Z 548.011,A -85,B 0,C 180,E1 -14490.004,E2 -14490.004} C_VEL
LIN {X 0,Y 332.244,Z 547.563,A -85,B 0,C 180,E1 -14491.216,E2 -14491.216} C_VEL
LIN {X 0,Y 332.126,Z 546.684,A -85,B 0,C 180,E1 -14492.43,E2 -14492.43} C_VEL
LIN {X 0,Y 332.083,Z 545.399,A -85,B 0,C 180,E1 -14493.645,E2 -14493.645} C_VEL
LIN {X 0,Y 332.106,Z 542.501,A -85,B 0,C 180,E1 -14495.537,E2 -14495.537} C_VEL
LIN {X 0,Y 332.252,Z 538.775,A -85,B 0,C 180,E1 -14497.296,E2 -14497.296} C_VEL
LIN {X 0,Y 332.511,Z 533.76,A -85,B 0,C 180,E1 -14499.125,E2 -14499.125} C_VEL
LIN {X 0,Y 332.92,Z 527.427,A -85,B 0,C 180,E1 -14500.956,E2 -14500.956} C_VEL
LIN {X 0,Y 333.801,Z 519.508,A -85,B 0,C 180,E1 -14502.776,E2 -14502.776} C_VEL
LIN {X 0,Y 334.764,Z 509.646,A -85,B 0,C 180,E1 -14504.596,E2 -14504.596} C_VEL
LIN {X 0,Y 335.681,Z 500.542,A -85,B 0,C 180,E1 -14505.954,E2 -14505.954} C_VEL
LIN {X 0,Y 336.825,Z 489.338,A -85,B 0,C 180,E1 -14507.301,E2 -14507.301} C_VEL
LIN {X 0,Y 337.498,Z 481.899,A -85,B 0,C 180,E1 -14508.048,E2 -14508.048} C_VEL
LIN {X 0,Y 336.547,Z 470.14,A -85,B 0,C 180,E1 -14509.075,E2 -14509.075} C_VEL
LIN {X 0,Y 334.987,Z 456.878,A -85,B 0,C 180,E1 -14509.993,E2 -14509.993} C_VEL
LIN {X 0,Y 333.034,Z 443.296,A -85,B 0,C 180,E1 -14510.689,E2 -14510.689} C_VEL
LIN {X 0,Y 332.874,Z 441.736,A -85,B 0,C 180,E1 -14510.795,E2 -14510.795} C_VEL
LIN {X 0,Y 333.523,Z 433.812,A -85,B 0,C 180,E1 -14515.027,E2 -14515.027} C_VEL
LIN {X 0,Y 334.275,Z 426.636,A -85,B 0,C 180,E1 -14518.923,E2 -14518.923} C_VEL
LIN {X 0,Y 335.112,Z 420.52,A -85,B 0,C 180,E1 -14522.325,E2 -14522.325} C_VEL
LIN {X 0,Y 335.997,Z 414.331,A -85,B 0,C 180,E1 -14525.855,E2 -14525.855} C_VEL
LIN {X 0,Y 335.721,Z 410.546,A -85,B 0,C 180,E1 -14528.142,E2 -14528.142} C_VEL
LIN {X 0,Y 334.986,Z 406.132,A -85,B 0,C 180,E1 -14530.949,E2 -14530.949} C_VEL
LIN {X 0,Y 334.071,Z 401.037,A -85,B 0,C 180,E1 -14534.333,E2 -14534.333} C_VEL
LIN {X 0,Y 333.659,Z 398.923,A -85,B 0,C 180,E1 -14535.839,E2 -14535.839} C_VEL
LIN {X 0,Y 333.618,Z 398.93,A -85,B 0,C 180,E1 -14539.326,E2 -14539.326} C_VEL
LIN {X 0,Y 333.677,Z 398.923,A -85,B 0,C 180,E1 -14543.17,E2 -14543.17} C_VEL
LIN {X 0,Y 333.688,Z 398.921,A -85,B 0,C 180,E1 -14545.342,E2 -14545.342} C_VEL
LIN {X 0,Y 333.644,Z 398.922,A -85,B 0,C 180,E1 -14548.222,E2 -14548.222} C_VEL
LIN {X 0,Y 333.669,Z 398.924,A -85,B 0,C 180,E1 -14551.023,E2 -14551.023} C_VEL
LIN {X 0,Y 333.712,Z 398.919,A -85,B 0,C 180,E1 -14555.089,E2 -14555.089} C_VEL
LIN {X 0,Y 333.674,Z 398.924,A -85,B 0,C 180,E1 -14559.018,E2 -14559.018} C_VEL
LIN {X 0,Y 333.756,Z 398.909,A -85,B 0,C 180,E1 -14561.586,E2 -14561.586} C_VEL
LIN {X 0,Y 333.825,Z 398.9,A -85,B 0,C 180,E1 -14565.577,E2 -14565.577} C_VEL
LIN {X 0,Y 333.831,Z 398.904,A -85,B 0,C 180,E1 -14569.077,E2 -14569.077} C_VEL
LIN {X 0,Y 334.004,Z 398.881,A -85,B 0,C 180,E1 -14572.746,E2 -14572.746} C_VEL
LIN {X 0,Y 333.812,Z 398.905,A -85,B 0,C 180,E1 -14575.168,E2 -14575.168} C_VEL
LIN {X 0,Y 334.116,Z 398.864,A -85,B 0,C 180,E1 -14577.588,E2 -14577.588} C_VEL
LIN {X 0,Y 334.201,Z 398.853,A -85,B 0,C 180,E1 -14579.999,E2 -14579.999} C_VEL
LIN {X 0,Y 334.085,Z 398.869,A -85,B 0,C 180,E1 -14582.41,E2 -14582.41} C_VEL
LIN {X 0,Y 333.97,Z 398.88,A -85,B 0,C 180,E1 -14586.548,E2 -14586.548} C_VEL
LIN {X 0,Y 333.833,Z 398.898,A -85,B 0,C 180,E1 -14589.695,E2 -14589.695} C_VEL
LIN {X 0,Y 333.805,Z 398.903,A -85,B 0,C 180,E1 -14593.39,E2 -14593.39} C_VEL
LIN {X 0,Y 333.731,Z 398.913,A -85,B 0,C 180,E1 -14597.146,E2 -14597.146} C_VEL
LIN {X 0,Y 333.676,Z 398.918,A -85,B 0,C 180,E1 -14599.693,E2 -14599.693} C_VEL
LIN {X 0,Y 333.68,Z 398.917,A -85,B 0,C 180,E1 -14603.588,E2 -14603.588} C_VEL
LIN {X 0,Y 333.74,Z 398.912,A -85,B 0,C 180,E1 -14606.245,E2 -14606.245} C_VEL
LIN {X 0,Y 333.69,Z 398.919,A -85,B 0,C 180,E1 -14608.973,E2 -14608.973} C_VEL
LIN {X 0,Y 333.646,Z 398.923,A -85,B 0,C 180,E1 -14613.206,E2 -14613.206} C_VEL
LIN {X 0,Y 333.684,Z 398.919,A -85,B 0,C 180,E1 -14616.136,E2 -14616.136} C_VEL
LIN {X 0,Y 333.641,Z 398.923,A -85,B 0,C 180,E1 -14619.191,E2 -14619.191} C_VEL
LIN {X 0,Y 333.64,Z 398.928,A -85,B 0,C 180,E1 -14622.497,E2 -14622.497} C_VEL
LIN {X 0,Y 333.602,Z 398.928,A -85,B 0,C 180,E1 -14625.952,E2 -14625.952} C_VEL
LIN {X 0,Y 333.652,Z 398.921,A -85,B 0,C 180,E1 -14629.312,E2 -14629.312} C_VEL
LIN {X 0,Y 333.669,Z 398.919,A -85,B 0,C 180,E1 -14633.165,E2 -14633.165} C_VEL
LIN {X 0,Y 333.678,Z 398.918,A -85,B 0,C 180,E1 -14635.338,E2 -14635.338} C_VEL
LIN {X 0,Y 333.694,Z 398.916,A -85,B 0,C 180,E1 -14639.633,E2 -14639.633} C_VEL
LIN {X 0,Y 333.742,Z 398.915,A -85,B 0,C 180,E1 -14642.397,E2 -14642.397} C_VEL
LIN {X 0,Y 333.729,Z 398.912,A -85,B 0,C 180,E1 -14645.087,E2 -14645.087} C_VEL
LIN {X 0,Y 333.68,Z 398.918,A -85,B 0,C 180,E1 -14649.015,E2 -14649.015} C_VEL
LIN {X 0,Y 333.793,Z 398.904,A -85,B 0,C 180,E1 -14651.585,E2 -14651.585} C_VEL
LIN {X 0,Y 333.807,Z 398.902,A -85,B 0,C 180,E1 -14655.573,E2 -14655.573} C_VEL
LIN {X 0,Y 333.831,Z 398.899,A -85,B 0,C 180,E1 -14659.074,E2 -14659.074} C_VEL
LIN {X 0,Y 334.001,Z 398.879,A -85,B 0,C 180,E1 -14662.743,E2 -14662.743} C_VEL
LIN {X 0,Y 333.802,Z 398.902,A -85,B 0,C 180,E1 -14665.165,E2 -14665.165} C_VEL
LIN {X 0,Y 334.098,Z 398.866,A -85,B 0,C 180,E1 -14667.584,E2 -14667.584} C_VEL
LIN {X 0,Y 334.238,Z 398.852,A -85,B 0,C 180,E1 -14669.996,E2 -14669.996} C_VEL
LIN {X 0,Y 334.099,Z 398.869,A -85,B 0,C 180,E1 -14672.407,E2 -14672.407} C_VEL
LIN {X 0,Y 334.015,Z 398.876,A -85,B 0,C 180,E1 -14677.248,E2 -14677.248} C_VEL
LIN {X 0,Y 333.825,Z 398.899,A -85,B 0,C 180,E1 -14680.917,E2 -14680.917} C_VEL
LIN {X 0,Y 333.794,Z 398.904,A -85,B 0,C 180,E1 -14684.63,E2 -14684.63} C_VEL
LIN {X 0,Y 333.781,Z 398.906,A -85,B 0,C 180,E1 -14688.651,E2 -14688.651} C_VEL
LIN {X 0,Y 333.673,Z 398.921,A -85,B 0,C 180,E1 -14692.274,E2 -14692.274} C_VEL
LIN {X 0,Y 333.656,Z 398.92,A -85,B 0,C 180,E1 -14695.081,E2 -14695.081} C_VEL
LIN {X 0,Y 333.463,Z 398.948,A -85,B 0,C 180,E1 -14697.729,E2 -14697.729} C_VEL
LIN {X 0,Y 333.154,Z 398.985,A -85,B 0,C 180,E1 -14700.411,E2 -14700.411} C_VEL
LIN {X 0,Y 332.739,Z 399.042,A -85,B 0,C 180,E1 -14703.303,E2 -14703.303} C_VEL
LIN {X 0,Y 332.64,Z 399.993,A -85,B 0,C 180,E1 -14704.775,E2 -14704.775} C_VEL
LIN {X 0,Y 332.553,Z 403.428,A -85,B 0,C 180,E1 -14708.564,E2 -14708.564} C_VEL
LIN {X 0,Y 332.483,Z 406.063,A -85,B 0,C 180,E1 -14711.386,E2 -14711.386} C_VEL
LIN {X 0,Y 335.759,Z 419.8,A -85,B 0,C 180,E1 -14712.203,E2 -14712.203} C_VEL
LIN {X 0,Y 338.252,Z 431.242,A -85,B 0,C 180,E1 -14713.066,E2 -14713.066} C_VEL
LIN {X 0,Y 339.069,Z 436.229,A -85,B 0,C 180,E1 -14713.495,E2 -14713.495} C_VEL
LIN {X 0,Y 338.119,Z 448.556,A -85,B 0,C 180,E1 -14714.612,E2 -14714.612} C_VEL
LIN {X 0,Y 336.981,Z 459.67,A -85,B 0,C 180,E1 -14715.89,E2 -14715.89} C_VEL
LIN {X 0,Y 335.936,Z 470.443,A -85,B 0,C 180,E1 -14717.436,E2 -14717.436} C_VEL
LIN {X 0,Y 334.951,Z 479.468,A -85,B 0,C 180,E1 -14719.048,E2 -14719.048} C_VEL
LIN {X 0,Y 334.047,Z 487.725,A -85,B 0,C 180,E1 -14720.865,E2 -14720.865} C_VEL
LIN {X 0,Y 333.317,Z 494.888,A -85,B 0,C 180,E1 -14722.846,E2 -14722.846} C_VEL
LIN {X 0,Y 332.899,Z 499.673,A -85,B 0,C 180,E1 -14724.511,E2 -14724.511} C_VEL
LIN {X 0,Y 332.491,Z 504.391,A -85,B 0,C 180,E1 -14726.664,E2 -14726.664} C_VEL
LIN {X 0,Y 332.211,Z 506.729,A -85,B 0,C 180,E1 -14728.072,E2 -14728.072} C_VEL
LIN {X 0,Y 332.069,Z 508.313,A -85,B 0,C 180,E1 -14729.385,E2 -14729.385} C_VEL
LIN {X 0,Y 331.365,Z 509.368,A -85,B 0,C 180,E1 -14730.381,E2 -14730.381} C_VEL
LIN {X 0,Y 328.467,Z 510.446,A -85,B 0,C 180,E1 -14732.019,E2 -14732.019} C_VEL
LIN {X 0,Y 326.077,Z 510.711,A -85,B 0,C 180,E1 -14733.354,E2 -14733.354} C_VEL
LIN {X 0,Y 325.118,Z 510.582,A -85,B 0,C 180,E1 -14734.387,E2 -14734.387} C_VEL
LIN {X 0,Y 325.074,Z 510.457,A -85,B 0,C 180,E1 -14734.736,E2 -14734.736} C_VEL
LIN {X 0,Y 325.547,Z 508.835,A -85,B 0,C 180,E1 -14737.135,E2 -14737.135} C_VEL
LIN {X 0,Y 326.093,Z 506.21,A -85,B 0,C 180,E1 -14739.17,E2 -14739.17} C_VEL
LIN {X 0,Y 326.755,Z 502.455,A -85,B 0,C 180,E1 -14741.179,E2 -14741.179} C_VEL
LIN {X 0,Y 327.714,Z 497.442,A -85,B 0,C 180,E1 -14743.172,E2 -14743.172} C_VEL
LIN {X 0,Y 328.951,Z 491.044,A -85,B 0,C 180,E1 -14745.146,E2 -14745.146} C_VEL
LIN {X 0,Y 330.423,Z 483.01,A -85,B 0,C 180,E1 -14747.097,E2 -14747.097} C_VEL
LIN {X 0,Y 331.936,Z 474.754,A -85,B 0,C 180,E1 -14748.707,E2 -14748.707} C_VEL
LIN {X 0,Y 333.402,Z 465.823,A -85,B 0,C 180,E1 -14750.139,E2 -14750.139} C_VEL
LIN {X 0,Y 335.069,Z 454.847,A -85,B 0,C 180,E1 -14751.558,E2 -14751.558} C_VEL
LIN {X 0,Y 336.575,Z 442.67,A -85,B 0,C 180,E1 -14752.804,E2 -14752.804} C_VEL
LIN {X 0,Y 334.328,Z 432.363,A -85,B 0,C 180,E1 -14753.968,E2 -14753.968} C_VEL
LIN {X 0,Y 330.439,Z 420.34,A -85,B 0,C 180,E1 -14755.235,E2 -14755.235} C_VEL
LIN {X 0,Y 327.025,Z 412.705,A -85,B 0,C 180,E1 -14756.035,E2 -14756.035} C_VEL
LIN {X 0,Y 326.368,Z 410.474,A -85,B 0,C 180,E1 -14756.258,E2 -14756.258} C_VEL
LIN {X 0,Y 327.132,Z 407.191,A -85,B 0,C 180,E1 -14761.232,E2 -14761.232} C_VEL
LIN {X 0,Y 327.244,Z 404.402,A -85,B 0,C 180,E1 -14766.165,E2 -14766.165} C_VEL
LIN {X 0,Y 327.313,Z 402.971,A -85,B 0,C 180,E1 -14769.036,E2 -14769.036} C_VEL
LIN {X 0,Y 327.003,Z 401.611,A -85,B 0,C 180,E1 -14772.412,E2 -14772.412} C_VEL
LIN {X 0,Y 326.88,Z 400.729,A -85,B 0,C 180,E1 -14774.953,E2 -14774.953} C_VEL
LIN {X 0,Y 326.733,Z 399.788,A -85,B 0,C 180,E1 -14778.857,E2 -14778.857} C_VEL
LIN {X 0,Y 326.658,Z 399.794,A -85,B 0,C 180,E1 -14782.786,E2 -14782.786} C_VEL
LIN {X 0,Y 326.657,Z 399.797,A -85,B 0,C 180,E1 -14786.861,E2 -14786.861} C_VEL
LIN {X 0,Y 326.633,Z 399.806,A -85,B 0,C 180,E1 -14789.663,E2 -14789.663} C_VEL
LIN {X 0,Y 326.746,Z 400.798,A -85,B 0,C 180,E1 -14792.992,E2 -14792.992} C_VEL
LIN {X 0,Y 326.96,Z 401.849,A -85,B 0,C 180,E1 -14795.477,E2 -14795.477} C_VEL
LIN {X 0,Y 327.376,Z 404.082,A -85,B 0,C 180,E1 -14799.4,E2 -14799.4} C_VEL
LIN {X 0,Y 327.722,Z 405.697,A -85,B 0,C 180,E1 -14801.668,E2 -14801.668} C_VEL
LIN {X 0,Y 328.186,Z 408.578,A -85,B 0,C 180,E1 -14805.042,E2 -14805.042} C_VEL
LIN {X 0,Y 328.802,Z 412.128,A -85,B 0,C 180,E1 -14808.508,E2 -14808.508} C_VEL
LIN {X 0,Y 329.421,Z 416.364,A -85,B 0,C 180,E1 -14812.128,E2 -14812.128} C_VEL
LIN {X 0,Y 329.4,Z 419.092,A -85,B 0,C 180,E1 -14814.171,E2 -14814.171} C_VEL
LIN {X 0,Y 328.323,Z 424.293,A -85,B 0,C 180,E1 -14817.653,E2 -14817.653} C_VEL
LIN {X 0,Y 327.251,Z 430.964,A -85,B 0,C 180,E1 -14821.811,E2 -14821.811} C_VEL
LIN {X 0,Y 326.536,Z 436.825,A -85,B 0,C 180,E1 -14825.247,E2 -14825.247} C_VEL
LIN {X 0,Y 326.481,Z 437.699,A -85,B 0,C 180,E1 -14825.747,E2 -14825.747} C_VEL
LIN {X 0,Y 327.334,Z 441.038,A -85,B 0,C 180,E1 -14825.977,E2 -14825.977} C_VEL
LIN {X 0,Y 330.643,Z 454.084,A -85,B 0,C 180,E1 -14827.033,E2 -14827.033} C_VEL
LIN {X 0,Y 332.647,Z 466.975,A -85,B 0,C 180,E1 -14828.177,E2 -14828.177} C_VEL
LIN {X 0,Y 333.373,Z 477.04,A -85,B 0,C 180,E1 -14829.166,E2 -14829.166} C_VEL
LIN {X 0,Y 333.281,Z 487.21,A -85,B 0,C 180,E1 -14830.287,E2 -14830.287} C_VEL
LIN {X 0,Y 331.546,Z 498.133,A -85,B 0,C 180,E1 -14831.625,E2 -14831.625} C_VEL
LIN {X 0,Y 329.723,Z 508.896,A -85,B 0,C 180,E1 -14833.282,E2 -14833.282} C_VEL
LIN {X 0,Y 328.417,Z 517.412,A -85,B 0,C 180,E1 -14834.897,E2 -14834.897} C_VEL
LIN {X 0,Y 327.255,Z 525.063,A -85,B 0,C 180,E1 -14836.657,E2 -14836.657} C_VEL
LIN {X 0,Y 326.32,Z 530.584,A -85,B 0,C 180,E1 -14838.199,E2 -14838.199} C_VEL
LIN {X 0,Y 325.645,Z 536.048,A -85,B 0,C 180,E1 -14840.063,E2 -14840.063} C_VEL
LIN {X 0,Y 325.224,Z 540.351,A -85,B 0,C 180,E1 -14841.93,E2 -14841.93} C_VEL
LIN {X 0,Y 324.968,Z 544.149,A -85,B 0,C 180,E1 -14844.178,E2 -14844.178} C_VEL
LIN {X 0,Y 324.972,Z 546.429,A -85,B 0,C 180,E1 -14846.285,E2 -14846.285} C_VEL
LIN {X 0,Y 325.104,Z 547.597,A -85,B 0,C 180,E1 -14848.766,E2 -14848.766} C_VEL
LIN {X 0,Y 325.212,Z 547.569,A -85,B 0,C 180,E1 -14850.005,E2 -14850.005} C_VEL
LIN {X 0,Y 325.166,Z 547.078,A -85,B 0,C 180,E1 -14851.243,E2 -14851.243} C_VEL
LIN {X 0,Y 325.034,Z 546.171,A -85,B 0,C 180,E1 -14852.483,E2 -14852.483} C_VEL
LIN {X 0,Y 325.01,Z 544.859,A -85,B 0,C 180,E1 -14853.724,E2 -14853.724} C_VEL
LIN {X 0,Y 325.051,Z 541.323,A -85,B 0,C 180,E1 -14855.963,E2 -14855.963} C_VEL
LIN {X 0,Y 325.235,Z 536.533,A -85,B 0,C 180,E1 -14858.079,E2 -14858.079} C_VEL
LIN {X 0,Y 325.597,Z 531.017,A -85,B 0,C 180,E1 -14859.948,E2 -14859.948} C_VEL
LIN {X 0,Y 326.178,Z 524.108,A -85,B 0,C 180,E1 -14861.816,E2 -14861.816} C_VEL
LIN {X 0,Y 326.945,Z 517.064,A -85,B 0,C 180,E1 -14863.365,E2 -14863.365} C_VEL
LIN {X 0,Y 327.791,Z 508.567,A -85,B 0,C 180,E1 -14864.913,E2 -14864.913} C_VEL
LIN {X 0,Y 328.959,Z 498.147,A -85,B 0,C 180,E1 -14866.448,E2 -14866.448} C_VEL
LIN {X 0,Y 330.054,Z 487.939,A -85,B 0,C 180,E1 -14867.668,E2 -14867.668} C_VEL
LIN {X 0,Y 330.478,Z 481.926,A -85,B 0,C 180,E1 -14868.285,E2 -14868.285} C_VEL
LIN {X 0,Y 329.482,Z 469.674,A -85,B 0,C 180,E1 -14869.386,E2 -14869.386} C_VEL
LIN {X 0,Y 327.973,Z 456.827,A -85,B 0,C 180,E1 -14870.3,E2 -14870.3} C_VEL
LIN {X 0,Y 326.081,Z 443.412,A -85,B 0,C 180,E1 -14871.017,E2 -14871.017} C_VEL
LIN {X 0,Y 325.824,Z 441.466,A -85,B 0,C 180,E1 -14871.101,E2 -14871.101} C_VEL
LIN {X 0,Y 326.502,Z 433.798,A -85,B 0,C 180,E1 -14875.302,E2 -14875.302} C_VEL
LIN {X 0,Y 327.37,Z 426.125,A -85,B 0,C 180,E1 -14879.593,E2 -14879.593} C_VEL
LIN {X 0,Y 328.289,Z 419.486,A -85,B 0,C 180,E1 -14883.392,E2 -14883.392} C_VEL
LIN {X 0,Y 328.898,Z 415.522,A -85,B 0,C 180,E1 -14885.707,E2 -14885.707} C_VEL
LIN {X 0,Y 328.796,Z 412.232,A -85,B 0,C 180,E1 -14887.732,E2 -14887.732} C_VEL
LIN {X 0,Y 327.857,Z 406.587,A -85,B 0,C 180,E1 -14891.385,E2 -14891.385} C_VEL
LIN {X 0,Y 326.849,Z 401.015,A -85,B 0,C 180,E1 -14895.205,E2 -14895.205} C_VEL
LIN {X 0,Y 326.616,Z 399.801,A -85,B 0,C 180,E1 -14896.156,E2 -14896.156} C_VEL
LIN {X 0,Y 326.572,Z 399.804,A -85,B 0,C 180,E1 -14899.787,E2 -14899.787} C_VEL
LIN {X 0,Y 326.641,Z 399.798,A -85,B 0,C 180,E1 -14902.953,E2 -14902.953} C_VEL
LIN {X 0,Y 326.622,Z 399.797,A -85,B 0,C 180,E1 -14905.981,E2 -14905.981} C_VEL
LIN {X 0,Y 326.627,Z 399.799,A -85,B 0,C 180,E1 -14909.398,E2 -14909.398} C_VEL
LIN {X 0,Y 326.63,Z 399.801,A -85,B 0,C 180,E1 -14913.136,E2 -14913.136} C_VEL
LIN {X 0,Y 326.648,Z 399.793,A -85,B 0,C 180,E1 -14915.87,E2 -14915.87} C_VEL
LIN {X 0,Y 326.631,Z 399.795,A -85,B 0,C 180,E1 -14919.862,E2 -14919.862} C_VEL
LIN {X 0,Y 326.724,Z 399.784,A -85,B 0,C 180,E1 -14923.76,E2 -14923.76} C_VEL
LIN {X 0,Y 326.772,Z 399.778,A -85,B 0,C 180,E1 -14926.314,E2 -14926.314} C_VEL
LIN {X 0,Y 326.798,Z 399.775,A -85,B 0,C 180,E1 -14930.092,E2 -14930.092} C_VEL
LIN {X 0,Y 326.972,Z 399.753,A -85,B 0,C 180,E1 -14933.829,E2 -14933.829} C_VEL
LIN {X 0,Y 327.056,Z 399.743,A -85,B 0,C 180,E1 -14937.536,E2 -14937.536} C_VEL
LIN {X 0,Y 327.154,Z 399.73,A -85,B 0,C 180,E1 -14939.999,E2 -14939.999} C_VEL
LIN {X 0,Y 327.029,Z 399.748,A -85,B 0,C 180,E1 -14942.462,E2 -14942.462} C_VEL
LIN {X 0,Y 326.932,Z 399.757,A -85,B 0,C 180,E1 -14946.538,E2 -14946.538} C_VEL
LIN {X 0,Y 326.796,Z 399.775,A -85,B 0,C 180,E1 -14949.906,E2 -14949.906} C_VEL
LIN {X 0,Y 326.769,Z 399.778,A -85,B 0,C 180,E1 -14953.684,E2 -14953.684} C_VEL
LIN {X 0,Y 326.675,Z 399.79,A -85,B 0,C 180,E1 -14957.528,E2 -14957.528} C_VEL
LIN {X 0,Y 326.627,Z 399.796,A -85,B 0,C 180,E1 -14961.455,E2 -14961.455} C_VEL
LIN {X 0,Y 326.7,Z 399.787,A -85,B 0,C 180,E1 -14965.481,E2 -14965.481} C_VEL
LIN {X 0,Y 326.655,Z 399.794,A -85,B 0,C 180,E1 -14968.249,E2 -14968.249} C_VEL
LIN {X 0,Y 326.584,Z 399.803,A -85,B 0,C 180,E1 -14971.095,E2 -14971.095} C_VEL
LIN {X 0,Y 326.616,Z 399.798,A -85,B 0,C 180,E1 -14974.017,E2 -14974.017} C_VEL
LIN {X 0,Y 326.632,Z 399.796,A -85,B 0,C 180,E1 -14977.234,E2 -14977.234} C_VEL
LIN {X 0,Y 326.583,Z 399.802,A -85,B 0,C 180,E1 -14981.127,E2 -14981.127} C_VEL
LIN {X 0,Y 326.534,Z 399.811,A -85,B 0,C 180,E1 -14984.739,E2 -14984.739} C_VEL
LIN {X 0,Y 326.582,Z 399.804,A -85,B 0,C 180,E1 -14988.151,E2 -14988.151} C_VEL
LIN {X 0,Y 326.602,Z 399.799,A -85,B 0,C 180,E1 -14991.384,E2 -14991.384} C_VEL
LIN {X 0,Y 326.624,Z 399.798,A -85,B 0,C 180,E1 -14994.848,E2 -14994.848} C_VEL
LIN {X 0,Y 326.612,Z 399.798,A -85,B 0,C 180,E1 -14997.452,E2 -14997.452} C_VEL
LIN {X 0,Y 326.651,Z 399.798,A -85,B 0,C 180,E1 -15000.336,E2 -15000.336} C_VEL
LIN {X 0,Y 326.692,Z 399.792,A -85,B 0,C 180,E1 -15004.512,E2 -15004.512} C_VEL
LIN {X 0,Y 326.646,Z 399.797,A -85,B 0,C 180,E1 -15008.541,E2 -15008.541} C_VEL
LIN {X 0,Y 326.745,Z 399.781,A -85,B 0,C 180,E1 -15011.173,E2 -15011.173} C_VEL
LIN {X 0,Y 326.762,Z 399.779,A -85,B 0,C 180,E1 -15015.429,E2 -15015.429} C_VEL
LIN {X 0,Y 326.767,Z 399.779,A -85,B 0,C 180,E1 -15018.835,E2 -15018.835} C_VEL
LIN {X 0,Y 326.954,Z 399.758,A -85,B 0,C 180,E1 -15022.585,E2 -15022.585} C_VEL
LIN {X 0,Y 326.769,Z 399.778,A -85,B 0,C 180,E1 -15025.06,E2 -15025.06} C_VEL
LIN {X 0,Y 327.039,Z 399.745,A -85,B 0,C 180,E1 -15027.532,E2 -15027.532} C_VEL
LIN {X 0,Y 327.19,Z 399.73,A -85,B 0,C 180,E1 -15029.995,E2 -15029.995} C_VEL
LIN {X 0,Y 327.039,Z 399.747,A -85,B 0,C 180,E1 -15032.459,E2 -15032.459} C_VEL
LIN {X 0,Y 326.986,Z 399.757,A -85,B 0,C 180,E1 -15036.165,E2 -15036.165} C_VEL
LIN {X 0,Y 326.903,Z 399.763,A -85,B 0,C 180,E1 -15038.651,E2 -15038.651} C_VEL
LIN {X 0,Y 326.726,Z 399.786,A -85,B 0,C 180,E1 -15042.417,E2 -15042.417} C_VEL
LIN {X 0,Y 326.74,Z 399.782,A -85,B 0,C 180,E1 -15044.953,E2 -15044.953} C_VEL
LIN {X 0,Y 326.717,Z 399.785,A -85,B 0,C 180,E1 -15048.834,E2 -15048.834} C_VEL
LIN {X 0,Y 326.599,Z 399.799,A -85,B 0,C 180,E1 -15052.783,E2 -15052.783} C_VEL
LIN {X 0,Y 326.578,Z 399.803,A -85,B 0,C 180,E1 -15055.487,E2 -15055.487} C_VEL
LIN {X 0,Y 326.331,Z 399.835,A -85,B 0,C 180,E1 -15058.275,E2 -15058.275} C_VEL
LIN {X 0,Y 325.988,Z 399.876,A -85,B 0,C 180,E1 -15061.153,E2 -15061.153} C_VEL
LIN {X 0,Y 325.597,Z 400.204,A -85,B 0,C 180,E1 -15064.133,E2 -15064.133} C_VEL
LIN {X 0,Y 325.517,Z 402.918,A -85,B 0,C 180,E1 -15067.188,E2 -15067.188} C_VEL
LIN {X 0,Y 325.421,Z 406.483,A -85,B 0,C 180,E1 -15071.046,E2 -15071.046} C_VEL
LIN {X 0,Y 328.345,Z 418.674,A -85,B 0,C 180,E1 -15071.768,E2 -15071.768} C_VEL
LIN {X 0,Y 331.201,Z 431.615,A -85,B 0,C 180,E1 -15072.76,E2 -15072.76} C_VEL
LIN {X 0,Y 332.142,Z 436.565,A -85,B 0,C 180,E1 -15073.202,E2 -15073.202} C_VEL
LIN {X 0,Y 331.274,Z 448.066,A -85,B 0,C 180,E1 -15074.256,E2 -15074.256} C_VEL
LIN {X 0,Y 330.122,Z 459.196,A -85,B 0,C 180,E1 -15075.54,E2 -15075.54} C_VEL
LIN {X 0,Y 329.047,Z 469.979,A -85,B 0,C 180,E1 -15077.095,E2 -15077.095} C_VEL
LIN {X 0,Y 328.178,Z 478.172,A -85,B 0,C 180,E1 -15078.541,E2 -15078.541} C_VEL
LIN {X 0,Y 327.18,Z 486.525,A -85,B 0,C 180,E1 -15080.338,E2 -15080.338} C_VEL
LIN {X 0,Y 326.481,Z 493.339,A -85,B 0,C 180,E1 -15082.159,E2 -15082.159} C_VEL
LIN {X 0,Y 325.847,Z 499.907,A -85,B 0,C 180,E1 -15084.386,E2 -15084.386} C_VEL
LIN {X 0,Y 325.431,Z 504.684,A -85,B 0,C 180,E1 -15086.587,E2 -15086.587} C_VEL
LIN {X 0,Y 325.037,Z 507.975,A -85,B 0,C 180,E1 -15088.741,E2 -15088.741} C_VEL
LIN {X 0,Y 324.919,Z 509.456,A -85,B 0,C 180,E1 -15090.167,E2 -15090.167} C_VEL
LIN {X 0,Y 324.931,Z 510.639,A -85,B 0,C 180,E1 -15092.46,E2 -15092.46} C_VEL
LIN {X 0,Y 325.074,Z 510.457,A -85,B 0,C 180,E1 -15094.736,E2 -15094.736} C_VEL
LIN {X 0,Y 324.574,Z 510.016,A -85,B 0,C 180,E1 -15095.772,E2 -15095.772} C_VEL
LIN {X 0,Y 322.108,Z 508.925,A -85,B 0,C 180,E1 -15097.463,E2 -15097.463} C_VEL
LIN {X 0,Y 320.077,Z 507.528,A -85,B 0,C 180,E1 -15098.816,E2 -15098.816} C_VEL
LIN {X 0,Y 319.348,Z 506.049,A -85,B 0,C 180,E1 -15099.837,E2 -15099.837} C_VEL
LIN {X 0,Y 319.366,Z 505.459,A -85,B 0,C 180,E1 -15100.176,E2 -15100.176} C_VEL
LIN {X 0,Y 320.109,Z 501.594,A -85,B 0,C 180,E1 -15102.1,E2 -15102.1} C_VEL
LIN {X 0,Y 321.316,Z 495.931,A -85,B 0,C 180,E1 -15104.213,E2 -15104.213} C_VEL
LIN {X 0,Y 322.681,Z 489.338,A -85,B 0,C 180,E1 -15106.139,E2 -15106.139} C_VEL
LIN {X 0,Y 323.971,Z 482.503,A -85,B 0,C 180,E1 -15107.762,E2 -15107.762} C_VEL
LIN {X 0,Y 325.613,Z 473.904,A -85,B 0,C 180,E1 -15109.43,E2 -15109.43} C_VEL
LIN {X 0,Y 327.323,Z 464.147,A -85,B 0,C 180,E1 -15110.954,E2 -15110.954} C_VEL
LIN {X 0,Y 328.973,Z 453.334,A -85,B 0,C 180,E1 -15112.328,E2 -15112.328} C_VEL
LIN {X 0,Y 330.167,Z 444.348,A -85,B 0,C 180,E1 -15113.26,E2 -15113.26} C_VEL
LIN {X 0,Y 327.992,Z 434.367,A -85,B 0,C 180,E1 -15114.454,E2 -15114.454} C_VEL
LIN {X 0,Y 324.648,Z 423.664,A -85,B 0,C 180,E1 -15115.656,E2 -15115.656} C_VEL
LIN {X 0,Y 320.451,Z 414.115,A -85,B 0,C 180,E1 -15116.74,E2 -15116.74} C_VEL
LIN {X 0,Y 319.328,Z 411.038,A -85,B 0,C 180,E1 -15117.084,E2 -15117.084} C_VEL
LIN {X 0,Y 320.14,Z 408.348,A -85,B 0,C 180,E1 -15121.259,E2 -15121.259} C_VEL
LIN {X 0,Y 320.265,Z 405.615,A -85,B 0,C 180,E1 -15126.3,E2 -15126.3} C_VEL
LIN {X 0,Y 320.32,Z 404.256,A -85,B 0,C 180,E1 -15129.172,E2 -15129.172} C_VEL
LIN {X 0,Y 320.03,Z 402.911,A -85,B 0,C 180,E1 -15132.687,E2 -15132.687} C_VEL
LIN {X 0,Y 319.906,Z 402.093,A -85,B 0,C 180,E1 -15135.286,E2 -15135.286} C_VEL
LIN {X 0,Y 319.753,Z 401.212,A -85,B 0,C 180,E1 -15139.251,E2 -15139.251} C_VEL
LIN {X 0,Y 319.637,Z 400.839,A -85,B 0,C 180,E1 -15143.315,E2 -15143.315} C_VEL
LIN {X 0,Y 319.628,Z 400.921,A -85,B 0,C 180,E1 -15146.09,E2 -15146.09} C_VEL
LIN {X 0,Y 319.681,Z 401.3,A -85,B 0,C 180,E1 -15148.926,E2 -15148.926} C_VEL
LIN {X 0,Y 319.763,Z 402.053,A -85,B 0,C 180,E1 -15151.837,E2 -15151.837} C_VEL
LIN {X 0,Y 320.068,Z 403.584,A -85,B 0,C 180,E1 -15155.676,E2 -15155.676} C_VEL
LIN {X 0,Y 320.497,Z 405.755,A -85,B 0,C 180,E1 -15159.49,E2 -15159.49} C_VEL
LIN {X 0,Y 320.948,Z 408.146,A -85,B 0,C 180,E1 -15162.753,E2 -15162.753} C_VEL
LIN {X 0,Y 321.432,Z 411.213,A -85,B 0,C 180,E1 -15166.182,E2 -15166.182} C_VEL
LIN {X 0,Y 322.057,Z 414.993,A -85,B 0,C 180,E1 -15169.8,E2 -15169.8} C_VEL
LIN {X 0,Y 322.459,Z 418.056,A -85,B 0,C 180,E1 -15172.399,E2 -15172.399} C_VEL
LIN {X 0,Y 322.246,Z 421.136,A -85,B 0,C 180,E1 -15174.701,E2 -15174.701} C_VEL
LIN {X 0,Y 320.991,Z 426.962,A -85,B 0,C 180,E1 -15178.639,E2 -15178.639} C_VEL
LIN {X 0,Y 320.058,Z 433.159,A -85,B 0,C 180,E1 -15182.546,E2 -15182.546} C_VEL
LIN {X 0,Y 319.546,Z 437.142,A -85,B 0,C 180,E1 -15184.933,E2 -15184.933} C_VEL
LIN {X 0,Y 320.462,Z 440.612,A -85,B 0,C 180,E1 -15185.203,E2 -15185.203} C_VEL
LIN {X 0,Y 323.817,Z 453.22,A -85,B 0,C 180,E1 -15186.296,E2 -15186.296} C_VEL
LIN {X 0,Y 325.952,Z 466.113,A -85,B 0,C 180,E1 -15187.489,E2 -15187.489} C_VEL
LIN {X 0,Y 326.76,Z 476.518,A -85,B 0,C 180,E1 -15188.559,E2 -15188.559} C_VEL
LIN {X 0,Y 326.646,Z 487.946,A -85,B 0,C 180,E1 -15189.869,E2 -15189.869} C_VEL
LIN {X 0,Y 324.677,Z 499.645,A -85,B 0,C 180,E1 -15191.386,E2 -15191.386} C_VEL
LIN {X 0,Y 322.928,Z 509.214,A -85,B 0,C 180,E1 -15192.919,E2 -15192.919} C_VEL
LIN {X 0,Y 321.563,Z 517.043,A -85,B 0,C 180,E1 -15194.448,E2 -15194.448} C_VEL
LIN {X 0,Y 320.56,Z 523.847,A -85,B 0,C 180,E1 -15196.05,E2 -15196.05} C_VEL
LIN {X 0,Y 319.348,Z 530.521,A -85,B 0,C 180,E1 -15197.937,E2 -15197.937} C_VEL
LIN {X 0,Y 318.608,Z 535.913,A -85,B 0,C 180,E1 -15199.841,E2 -15199.841} C_VEL
LIN {X 0,Y 318.171,Z 540.154,A -85,B 0,C 180,E1 -15201.75,E2 -15201.75} C_VEL
LIN {X 0,Y 317.915,Z 543.344,A -85,B 0,C 180,E1 -15203.659,E2 -15203.659} C_VEL
LIN {X 0,Y 317.849,Z 544.925,A -85,B 0,C 180,E1 -15204.931,E2 -15204.931} C_VEL
LIN {X 0,Y 317.897,Z 546.079,A -85,B 0,C 180,E1 -15206.202,E2 -15206.202} C_VEL
LIN {X 0,Y 318.008,Z 547.191,A -85,B 0,C 180,E1 -15208.738,E2 -15208.738} C_VEL
LIN {X 0,Y 318.135,Z 547.113,A -85,B 0,C 180,E1 -15210.005,E2 -15210.005} C_VEL
LIN {X 0,Y 318.073,Z 546.592,A -85,B 0,C 180,E1 -15211.271,E2 -15211.271} C_VEL
LIN {X 0,Y 317.943,Z 545.659,A -85,B 0,C 180,E1 -15212.538,E2 -15212.538} C_VEL
LIN {X 0,Y 317.938,Z 544.318,A -85,B 0,C 180,E1 -15213.807,E2 -15213.807} C_VEL
LIN {X 0,Y 317.961,Z 541.032,A -85,B 0,C 180,E1 -15215.922,E2 -15215.922} C_VEL
LIN {X 0,Y 318.096,Z 537.44,A -85,B 0,C 180,E1 -15217.622,E2 -15217.622} C_VEL
LIN {X 0,Y 318.487,Z 531.261,A -85,B 0,C 180,E1 -15219.851,E2 -15219.851} C_VEL
LIN {X 0,Y 319.041,Z 524.492,A -85,B 0,C 180,E1 -15221.761,E2 -15221.761} C_VEL
LIN {X 0,Y 319.956,Z 516.099,A -85,B 0,C 180,E1 -15223.663,E2 -15223.663} C_VEL
LIN {X 0,Y 320.771,Z 507.44,A -85,B 0,C 180,E1 -15225.247,E2 -15225.247} C_VEL
LIN {X 0,Y 322.078,Z 496.9,A -85,B 0,C 180,E1 -15226.81,E2 -15226.81} C_VEL
LIN {X 0,Y 323.212,Z 486.528,A -85,B 0,C 180,E1 -15228.055,E2 -15228.055} C_VEL
LIN {X 0,Y 323.462,Z 481.938,A -85,B 0,C 180,E1 -15228.532,E2 -15228.532} C_VEL
LIN {X 0,Y 322.548,Z 470.565,A -85,B 0,C 180,E1 -15229.601,E2 -15229.601} C_VEL
LIN {X 0,Y 320.981,Z 457.207,A -85,B 0,C 180,E1 -15230.595,E2 -15230.595} C_VEL
LIN {X 0,Y 319.121,Z 443.645,A -85,B 0,C 180,E1 -15231.354,E2 -15231.354} C_VEL
LIN {X 0,Y 318.787,Z 441.117,A -85,B 0,C 180,E1 -15231.463,E2 -15231.463} C_VEL
LIN {X 0,Y 319.456,Z 433.815,A -85,B 0,C 180,E1 -15235.576,E2 -15235.576} C_VEL
LIN {X 0,Y 320.284,Z 426.803,A -85,B 0,C 180,E1 -15239.59,E2 -15239.59} C_VEL
LIN {X 0,Y 321.166,Z 420.693,A -85,B 0,C 180,E1 -15243.17,E2 -15243.17} C_VEL
LIN {X 0,Y 321.877,Z 415.776,A -85,B 0,C 180,E1 -15246.128,E2 -15246.128} C_VEL
LIN {X 0,Y 321.671,Z 412.592,A -85,B 0,C 180,E1 -15248.135,E2 -15248.135} C_VEL
LIN {X 0,Y 320.94,Z 408.167,A -85,B 0,C 180,E1 -15251.072,E2 -15251.072} C_VEL
LIN {X 0,Y 320.022,Z 403.003,A -85,B 0,C 180,E1 -15254.653,E2 -15254.653} C_VEL
LIN {X 0,Y 319.566,Z 400.679,A -85,B 0,C 180,E1 -15256.473,E2 -15256.473} C_VEL
LIN {X 0,Y 319.561,Z 400.676,A -85,B 0,C 180,E1 -15260.372,E2 -15260.372} C_VEL
LIN {X 0,Y 319.594,Z 400.672,A -85,B 0,C 180,E1 -15264.459,E2 -15264.459} C_VEL
LIN {X 0,Y 319.54,Z 400.678,A -85,B 0,C 180,E1 -15268.138,E2 -15268.138} C_VEL
LIN {X 0,Y 319.588,Z 400.674,A -85,B 0,C 180,E1 -15271.604,E2 -15271.604} C_VEL
LIN {X 0,Y 319.59,Z 400.676,A -85,B 0,C 180,E1 -15275.302,E2 -15275.302} C_VEL
LIN {X 0,Y 319.581,Z 400.673,A -85,B 0,C 180,E1 -15278.046,E2 -15278.046} C_VEL
LIN {X 0,Y 319.63,Z 400.667,A -85,B 0,C 180,E1 -15282.07,E2 -15282.07} C_VEL
LIN {X 0,Y 319.747,Z 400.653,A -85,B 0,C 180,E1 -15286.007,E2 -15286.007} C_VEL
LIN {X 0,Y 319.751,Z 400.652,A -85,B 0,C 180,E1 -15289.872,E2 -15289.872} C_VEL
LIN {X 0,Y 319.93,Z 400.63,A -85,B 0,C 180,E1 -15293.693,E2 -15293.693} C_VEL
LIN {X 0,Y 320,Z 400.622,A -85,B 0,C 180,E1 -15297.481,E2 -15297.481} C_VEL
LIN {X 0,Y 320.109,Z 400.608,A -85,B 0,C 180,E1 -15299.999,E2 -15299.999} C_VEL
LIN {X 0,Y 319.975,Z 400.627,A -85,B 0,C 180,E1 -15302.517,E2 -15302.517} C_VEL
LIN {X 0,Y 319.894,Z 400.634,A -85,B 0,C 180,E1 -15306.521,E2 -15306.521} C_VEL
LIN {X 0,Y 319.748,Z 400.653,A -85,B 0,C 180,E1 -15310.126,E2 -15310.126} C_VEL
LIN {X 0,Y 319.744,Z 400.653,A -85,B 0,C 180,E1 -15313.99,E2 -15313.99} C_VEL
LIN {X 0,Y 319.626,Z 400.668,A -85,B 0,C 180,E1 -15317.928,E2 -15317.928} C_VEL
LIN {X 0,Y 319.579,Z 400.674,A -85,B 0,C 180,E1 -15321.952,E2 -15321.952} C_VEL
LIN {X 0,Y 319.626,Z 400.669,A -85,B 0,C 180,E1 -15326.087,E2 -15326.087} C_VEL
LIN {X 0,Y 319.578,Z 400.677,A -85,B 0,C 180,E1 -15328.933,E2 -15328.933} C_VEL
LIN {X 0,Y 319.534,Z 400.679,A -85,B 0,C 180,E1 -15331.86,E2 -15331.86} C_VEL
LIN {X 0,Y 319.588,Z 400.673,A -85,B 0,C 180,E1 -15335.54,E2 -15335.54} C_VEL
LIN {X 0,Y 319.568,Z 400.675,A -85,B 0,C 180,E1 -15339.666,E2 -15339.666} C_VEL
LIN {X 0,Y 319.528,Z 400.68,A -85,B 0,C 180,E1 -15343.457,E2 -15343.457} C_VEL
LIN {X 0,Y 319.56,Z 400.677,A -85,B 0,C 180,E1 -15347.013,E2 -15347.013} C_VEL
LIN {X 0,Y 319.552,Z 400.681,A -85,B 0,C 180,E1 -15350.367,E2 -15350.367} C_VEL
LIN {X 0,Y 319.585,Z 400.679,A -85,B 0,C 180,E1 -15354.453,E2 -15354.453} C_VEL
LIN {X 0,Y 319.534,Z 400.682,A -85,B 0,C 180,E1 -15358.134,E2 -15358.134} C_VEL
LIN {X 0,Y 319.614,Z 400.669,A -85,B 0,C 180,E1 -15361.586,E2 -15361.586} C_VEL
LIN {X 0,Y 319.607,Z 400.67,A -85,B 0,C 180,E1 -15365.3,E2 -15365.3} C_VEL
LIN {X 0,Y 319.598,Z 400.674,A -85,B 0,C 180,E1 -15368.044,E2 -15368.044} C_VEL
LIN {X 0,Y 319.689,Z 400.661,A -85,B 0,C 180,E1 -15370.958,E2 -15370.958} C_VEL
LIN {X 0,Y 319.73,Z 400.655,A -85,B 0,C 180,E1 -15375.272,E2 -15375.272} C_VEL
LIN {X 0,Y 319.75,Z 400.655,A -85,B 0,C 180,E1 -15379.868,E2 -15379.868} C_VEL
LIN {X 0,Y 319.908,Z 400.636,A -85,B 0,C 180,E1 -15382.421,E2 -15382.421} C_VEL
LIN {X 0,Y 319.738,Z 400.654,A -85,B 0,C 180,E1 -15384.951,E2 -15384.951} C_VEL
LIN {X 0,Y 319.983,Z 400.624,A -85,B 0,C 180,E1 -15387.478,E2 -15387.478} C_VEL
LIN {X 0,Y 320.141,Z 400.608,A -85,B 0,C 180,E1 -15389.995,E2 -15389.995} C_VEL
LIN {X 0,Y 319.983,Z 400.626,A -85,B 0,C 180,E1 -15392.513,E2 -15392.513} C_VEL
LIN {X 0,Y 319.942,Z 400.632,A -85,B 0,C 180,E1 -15396.301,E2 -15396.301} C_VEL
LIN {X 0,Y 319.832,Z 400.642,A -85,B 0,C 180,E1 -15398.843,E2 -15398.843} C_VEL
LIN {X 0,Y 319.672,Z 400.663,A -85,B 0,C 180,E1 -15402.695,E2 -15402.695} C_VEL
LIN {X 0,Y 319.685,Z 400.661,A -85,B 0,C 180,E1 -15405.291,E2 -15405.291} C_VEL
LIN {X 0,Y 319.658,Z 400.664,A -85,B 0,C 180,E1 -15409.25,E2 -15409.25} C_VEL
LIN {X 0,Y 319.542,Z 400.679,A -85,B 0,C 180,E1 -15413.316,E2 -15413.316} C_VEL
LIN {X 0,Y 319.495,Z 400.689,A -85,B 0,C 180,E1 -15416.094,E2 -15416.094} C_VEL
LIN {X 0,Y 319.192,Z 400.722,A -85,B 0,C 180,E1 -15418.967,E2 -15418.967} C_VEL
LIN {X 0,Y 318.829,Z 400.773,A -85,B 0,C 180,E1 -15421.934,E2 -15421.934} C_VEL
LIN {X 0,Y 318.619,Z 400.8,A -85,B 0,C 180,E1 -15423.459,E2 -15423.459} C_VEL
LIN {X 0,Y 318.503,Z 401.975,A -85,B 0,C 180,E1 -15425.273,E2 -15425.273} C_VEL
LIN {X 0,Y 318.41,Z 404.519,A -85,B 0,C 180,E1 -15428.164,E2 -15428.164} C_VEL
LIN {X 0,Y 318.369,Z 406.805,A -85,B 0,C 180,E1 -15430.678,E2 -15430.678} C_VEL
LIN {X 0,Y 321.864,Z 421.509,A -85,B 0,C 180,E1 -15431.598,E2 -15431.598} C_VEL
LIN {X 0,Y 324.469,Z 433.512,A -85,B 0,C 180,E1 -15432.573,E2 -15432.573} C_VEL
LIN {X 0,Y 325.221,Z 438.942,A -85,B 0,C 180,E1 -15433.073,E2 -15433.073} C_VEL
LIN {X 0,Y 324.088,Z 451.441,A -85,B 0,C 180,E1 -15434.308,E2 -15434.308} C_VEL
LIN {X 0,Y 322.924,Z 462.21,A -85,B 0,C 180,E1 -15435.643,E2 -15435.643} C_VEL
LIN {X 0,Y 321.889,Z 472.225,A -85,B 0,C 180,E1 -15437.192,E2 -15437.192} C_VEL
LIN {X 0,Y 320.791,Z 481.283,A -85,B 0,C 180,E1 -15438.911,E2 -15438.911} C_VEL
LIN {X 0,Y 319.864,Z 489.449,A -85,B 0,C 180,E1 -15440.827,E2 -15440.827} C_VEL
LIN {X 0,Y 319.115,Z 496.54,A -85,B 0,C 180,E1 -15442.947,E2 -15442.947} C_VEL
LIN {X 0,Y 318.588,Z 501.897,A -85,B 0,C 180,E1 -15445.003,E2 -15445.003} C_VEL
LIN {X 0,Y 318.257,Z 505.906,A -85,B 0,C 180,E1 -15447.039,E2 -15447.039} C_VEL
LIN {X 0,Y 317.87,Z 509.239,A -85,B 0,C 180,E1 -15449.561,E2 -15449.561} C_VEL
LIN {X 0,Y 317.828,Z 510.333,A -85,B 0,C 180,E1 -15450.892,E2 -15450.892} C_VEL
LIN {X 0,Y 317.846,Z 511.016,A -85,B 0,C 180,E1 -15452.334,E2 -15452.334} C_VEL
LIN {X 0,Y 317.992,Z 510.94,A -85,B 0,C 180,E1 -15454.773,E2 -15454.773} C_VEL
LIN {X 0,Y 318.345,Z 509.951,A -85,B 0,C 180,E1 -15456.587,E2 -15456.587} C_VEL
LIN {X 0,Y 318.673,Z 508.617,A -85,B 0,C 180,E1 -15457.982,E2 -15457.982} C_VEL
LIN {X 0,Y 319.366,Z 505.459,A -85,B 0,C 180,E1 -15460.176,E2 -15460.176} C_VEL
LIN {X 0,Y 319.048,Z 503.685,A -85,B 0,C 180,E1 -15461.184,E2 -15461.184} C_VEL
LIN {X 0,Y 316.944,Z 500.485,A -85,B 0,C 180,E1 -15462.839,E2 -15462.839} C_VEL
LIN {X 0,Y 315.057,Z 496.725,A -85,B 0,C 180,E1 -15464.465,E2 -15464.465} C_VEL
LIN {X 0,Y 315.068,Z 493.937,A -85,B 0,C 180,E1 -15465.41,E2 -15465.41} C_VEL
LIN {X 0,Y 316.695,Z 486.176,A -85,B 0,C 180,E1 -15467.507,E2 -15467.507} C_VEL
LIN {X 0,Y 318.313,Z 478.452,A -85,B 0,C 180,E1 -15469.184,E2 -15469.184} C_VEL
LIN {X 0,Y 319.984,Z 469.651,A -85,B 0,C 180,E1 -15470.753,E2 -15470.753} C_VEL
LIN {X 0,Y 321.932,Z 458.672,A -85,B 0,C 180,E1 -15472.317,E2 -15472.317} C_VEL
LIN {X 0,Y 323.684,Z 447.286,A -85,B 0,C 180,E1 -15473.612,E2 -15473.612} C_VEL
LIN {X 0,Y 323.519,Z 444.668,A -85,B 0,C 180,E1 -15473.918,E2 -15473.918} C_VEL
LIN {X 0,Y 320.966,Z 433.721,A -85,B 0,C 180,E1 -15475.292,E2 -15475.292} C_VEL
LIN {X 0,Y 318.094,Z 424.942,A -85,B 0,C 180,E1 -15476.344,E2 -15476.344} C_VEL
LIN {X 0,Y 313.529,Z 414.847,A -85,B 0,C 180,E1 -15477.572,E2 -15477.572} C_VEL
LIN {X 0,Y 312.41,Z 411.655,A -85,B 0,C 180,E1 -15477.906,E2 -15477.906} C_VEL
LIN {X 0,Y 313.145,Z 409.548,A -85,B 0,C 180,E1 -15481.287,E2 -15481.287} C_VEL
LIN {X 0,Y 313.285,Z 406.828,A -85,B 0,C 180,E1 -15486.441,E2 -15486.441} C_VEL
LIN {X 0,Y 313.338,Z 405.535,A -85,B 0,C 180,E1 -15489.327,E2 -15489.327} C_VEL
LIN {X 0,Y 313.039,Z 404.229,A -85,B 0,C 180,E1 -15492.975,E2 -15492.975} C_VEL
LIN {X 0,Y 312.928,Z 403.463,A -85,B 0,C 180,E1 -15495.636,E2 -15495.636} C_VEL
LIN {X 0,Y 312.786,Z 402.687,A -85,B 0,C 180,E1 -15499.697,E2 -15499.697} C_VEL
LIN {X 0,Y 312.713,Z 402.431,A -85,B 0,C 180,E1 -15503.863,E2 -15503.863} C_VEL
LIN {X 0,Y 312.731,Z 402.614,A -85,B 0,C 180,E1 -15506.71,E2 -15506.71} C_VEL
LIN {X 0,Y 312.789,Z 403.106,A -85,B 0,C 180,E1 -15509.626,E2 -15509.626} C_VEL
LIN {X 0,Y 313.005,Z 404.425,A -85,B 0,C 180,E1 -15513.833,E2 -15513.833} C_VEL
LIN {X 0,Y 313.274,Z 406.074,A -85,B 0,C 180,E1 -15517.282,E2 -15517.282} C_VEL
LIN {X 0,Y 313.706,Z 408.075,A -85,B 0,C 180,E1 -15520.52,E2 -15520.52} C_VEL
LIN {X 0,Y 314.181,Z 410.664,A -85,B 0,C 180,E1 -15523.905,E2 -15523.905} C_VEL
LIN {X 0,Y 314.805,Z 414.457,A -85,B 0,C 180,E1 -15527.96,E2 -15527.96} C_VEL
LIN {X 0,Y 315.369,Z 418.203,A -85,B 0,C 180,E1 -15531.4,E2 -15531.4} C_VEL
LIN {X 0,Y 315.464,Z 420.566,A -85,B 0,C 180,E1 -15533.325,E2 -15533.325} C_VEL
LIN {X 0,Y 314.927,Z 423.738,A -85,B 0,C 180,E1 -15535.661,E2 -15535.661} C_VEL
LIN {X 0,Y 313.679,Z 429.735,A -85,B 0,C 180,E1 -15539.734,E2 -15539.734} C_VEL
LIN {X 0,Y 312.691,Z 436.643,A -85,B 0,C 180,E1 -15544.095,E2 -15544.095} C_VEL
LIN {X 0,Y 313.619,Z 440.119,A -85,B 0,C 180,E1 -15544.37,E2 -15544.37} C_VEL
LIN {X 0,Y 317.058,Z 452.766,A -85,B 0,C 180,E1 -15545.535,E2 -15545.535} C_VEL
LIN {X 0,Y 319.093,Z 464.122,A -85,B 0,C 180,E1 -15546.649,E2 -15546.649} C_VEL
LIN {X 0,Y 320.209,Z 475.851,A -85,B 0,C 180,E1 -15547.894,E2 -15547.894} C_VEL
LIN {X 0,Y 320.153,Z 487.487,A -85,B 0,C 180,E1 -15549.275,E2 -15549.275} C_VEL
LIN {X 0,Y 318.369,Z 498.051,A -85,B 0,C 180,E1 -15550.668,E2 -15550.668} C_VEL
LIN {X 0,Y 316.49,Z 507.755,A -85,B 0,C 180,E1 -15552.227,E2 -15552.227} C_VEL
LIN {X 0,Y 314.904,Z 516.118,A -85,B 0,C 180,E1 -15553.861,E2 -15553.861} C_VEL
LIN {X 0,Y 313.672,Z 523.947,A -85,B 0,C 180,E1 -15555.737,E2 -15555.737} C_VEL
LIN {X 0,Y 312.39,Z 530.5,A -85,B 0,C 180,E1 -15557.664,E2 -15557.664} C_VEL
LIN {X 0,Y 311.588,Z 535.775,A -85,B 0,C 180,E1 -15559.61,E2 -15559.61} C_VEL
LIN {X 0,Y 311.113,Z 539.937,A -85,B 0,C 180,E1 -15561.562,E2 -15561.562} C_VEL
LIN {X 0,Y 310.835,Z 543.078,A -85,B 0,C 180,E1 -15563.514,E2 -15563.514} C_VEL
LIN {X 0,Y 310.8,Z 545.731,A -85,B 0,C 180,E1 -15566.115,E2 -15566.115} C_VEL
LIN {X 0,Y 310.801,Z 546.456,A -85,B 0,C 180,E1 -15567.413,E2 -15567.413} C_VEL
LIN {X 0,Y 310.913,Z 546.774,A -85,B 0,C 180,E1 -15568.71,E2 -15568.71} C_VEL
LIN {X 0,Y 311.06,Z 546.645,A -85,B 0,C 180,E1 -15570.005,E2 -15570.005} C_VEL
LIN {X 0,Y 310.98,Z 546.094,A -85,B 0,C 180,E1 -15571.3,E2 -15571.3} C_VEL
LIN {X 0,Y 310.857,Z 545.133,A -85,B 0,C 180,E1 -15572.596,E2 -15572.596} C_VEL
LIN {X 0,Y 310.869,Z 543.744,A -85,B 0,C 180,E1 -15573.894,E2 -15573.894} C_VEL
LIN {X 0,Y 310.888,Z 540.669,A -85,B 0,C 180,E1 -15575.908,E2 -15575.908} C_VEL
LIN {X 0,Y 311.027,Z 536.743,A -85,B 0,C 180,E1 -15577.797,E2 -15577.797} C_VEL
LIN {X 0,Y 311.457,Z 530.477,A -85,B 0,C 180,E1 -15580.076,E2 -15580.076} C_VEL
LIN {X 0,Y 312.053,Z 523.631,A -85,B 0,C 180,E1 -15582.029,E2 -15582.029} C_VEL
LIN {X 0,Y 312.854,Z 516.659,A -85,B 0,C 180,E1 -15583.648,E2 -15583.648} C_VEL
LIN {X 0,Y 313.669,Z 508.718,A -85,B 0,C 180,E1 -15585.183,E2 -15585.183} C_VEL
LIN {X 0,Y 314.84,Z 499.248,A -85,B 0,C 180,E1 -15586.69,E2 -15586.69} C_VEL
LIN {X 0,Y 316.133,Z 487.908,A -85,B 0,C 180,E1 -15588.138,E2 -15588.138} C_VEL
LIN {X 0,Y 316.451,Z 481.95,A -85,B 0,C 180,E1 -15588.79,E2 -15588.79} C_VEL
LIN {X 0,Y 315.405,Z 469.399,A -85,B 0,C 180,E1 -15589.993,E2 -15589.993} C_VEL
LIN {X 0,Y 313.864,Z 455.955,A -85,B 0,C 180,E1 -15590.998,E2 -15590.998} C_VEL
LIN {X 0,Y 312.042,Z 442.935,A -85,B 0,C 180,E1 -15591.731,E2 -15591.731} C_VEL
LIN {X 0,Y 311.736,Z 440.742,A -85,B 0,C 180,E1 -15591.843,E2 -15591.843} C_VEL
LIN {X 0,Y 312.407,Z 433.803,A -85,B 0,C 180,E1 -15595.86,E2 -15595.86} C_VEL
LIN {X 0,Y 313.197,Z 427.465,A -85,B 0,C 180,E1 -15599.586,E2 -15599.586} C_VEL
LIN {X 0,Y 314.127,Z 421.377,A -85,B 0,C 180,E1 -15603.244,E2 -15603.244} C_VEL
LIN {X 0,Y 314.725,Z 417.693,A -85,B 0,C 180,E1 -15605.497,E2 -15605.497} C_VEL
LIN {X 0,Y 314.74,Z 414.089,A -85,B 0,C 180,E1 -15607.796,E2 -15607.796} C_VEL
LIN {X 0,Y 313.866,Z 408.845,A -85,B 0,C 180,E1 -15611.347,E2 -15611.347} C_VEL
LIN {X 0,Y 312.94,Z 403.776,A -85,B 0,C 180,E1 -15614.973,E2 -15614.973} C_VEL
LIN {X 0,Y 312.55,Z 401.554,A -85,B 0,C 180,E1 -15616.783,E2 -15616.783} C_VEL
LIN {X 0,Y 312.51,Z 401.558,A -85,B 0,C 180,E1 -15620.972,E2 -15620.972} C_VEL
LIN {X 0,Y 312.546,Z 401.55,A -85,B 0,C 180,E1 -15624.221,E2 -15624.221} C_VEL
LIN {X 0,Y 312.518,Z 401.557,A -85,B 0,C 180,E1 -15627.334,E2 -15627.334} C_VEL
LIN {X 0,Y 312.523,Z 401.557,A -85,B 0,C 180,E1 -15631.293,E2 -15631.293} C_VEL
LIN {X 0,Y 312.564,Z 401.549,A -85,B 0,C 180,E1 -15634.708,E2 -15634.708} C_VEL
LIN {X 0,Y 312.537,Z 401.555,A -85,B 0,C 180,E1 -15638.912,E2 -15638.912} C_VEL
LIN {X 0,Y 312.594,Z 401.549,A -85,B 0,C 180,E1 -15643.005,E2 -15643.005} C_VEL
LIN {X 0,Y 312.701,Z 401.531,A -85,B 0,C 180,E1 -15645.685,E2 -15645.685} C_VEL
LIN {X 0,Y 312.701,Z 401.531,A -85,B 0,C 180,E1 -15649.641,E2 -15649.641} C_VEL
LIN {X 0,Y 312.844,Z 401.513,A -85,B 0,C 180,E1 -15652.252,E2 -15652.252} C_VEL
LIN {X 0,Y 312.718,Z 401.533,A -85,B 0,C 180,E1 -15654.841,E2 -15654.841} C_VEL
LIN {X 0,Y 312.999,Z 401.497,A -85,B 0,C 180,E1 -15658.712,E2 -15658.712} C_VEL
LIN {X 0,Y 312.997,Z 401.496,A -85,B 0,C 180,E1 -15661.285,E2 -15661.285} C_VEL
LIN {X 0,Y 312.708,Z 401.532,A -85,B 0,C 180,E1 -15665.157,E2 -15665.157} C_VEL
LIN {X 0,Y 312.81,Z 401.517,A -85,B 0,C 180,E1 -15667.746,E2 -15667.746} C_VEL
LIN {X 0,Y 312.675,Z 401.534,A -85,B 0,C 180,E1 -15671.67,E2 -15671.67} C_VEL
LIN {X 0,Y 312.681,Z 401.538,A -85,B 0,C 180,E1 -15674.862,E2 -15674.862} C_VEL
LIN {X 0,Y 312.56,Z 401.55,A -85,B 0,C 180,E1 -15679.19,E2 -15679.19} C_VEL
LIN {X 0,Y 312.538,Z 401.555,A -85,B 0,C 180,E1 -15682.778,E2 -15682.778} C_VEL
LIN {X 0,Y 312.606,Z 401.543,A -85,B 0,C 180,E1 -15685.93,E2 -15685.93} C_VEL
LIN {X 0,Y 312.518,Z 401.553,A -85,B 0,C 180,E1 -15689.651,E2 -15689.651} C_VEL
LIN {X 0,Y 312.53,Z 401.552,A -85,B 0,C 180,E1 -15693.686,E2 -15693.686} C_VEL
LIN {X 0,Y 312.524,Z 401.553,A -85,B 0,C 180,E1 -15697.384,E2 -15697.384} C_VEL
LIN {X 0,Y 312.497,Z 401.56,A -85,B 0,C 180,E1 -15700.706,E2 -15700.706} C_VEL
LIN {X 0,Y 312.459,Z 401.563,A -85,B 0,C 180,E1 -15704.206,E2 -15704.206} C_VEL
LIN {X 0,Y 312.474,Z 401.559,A -85,B 0,C 180,E1 -15707.919,E2 -15707.919} C_VEL
LIN {X 0,Y 312.504,Z 401.557,A -85,B 0,C 180,E1 -15710.967,E2 -15710.967} C_VEL
LIN {X 0,Y 312.537,Z 401.554,A -85,B 0,C 180,E1 -15714.217,E2 -15714.217} C_VEL
LIN {X 0,Y 312.508,Z 401.554,A -85,B 0,C 180,E1 -15717.33,E2 -15717.33} C_VEL
LIN {X 0,Y 312.547,Z 401.55,A -85,B 0,C 180,E1 -15721.275,E2 -15721.275} C_VEL
LIN {X 0,Y 312.588,Z 401.547,A -85,B 0,C 180,E1 -15724.707,E2 -15724.707} C_VEL
LIN {X 0,Y 312.589,Z 401.545,A -85,B 0,C 180,E1 -15727.525,E2 -15727.525} C_VEL
LIN {X 0,Y 312.638,Z 401.539,A -85,B 0,C 180,E1 -15731.652,E2 -15731.652} C_VEL
LIN {X 0,Y 312.692,Z 401.532,A -85,B 0,C 180,E1 -15735.682,E2 -15735.682} C_VEL
LIN {X 0,Y 312.696,Z 401.532,A -85,B 0,C 180,E1 -15739.637,E2 -15739.637} C_VEL
LIN {X 0,Y 312.849,Z 401.517,A -85,B 0,C 180,E1 -15742.249,E2 -15742.249} C_VEL
LIN {X 0,Y 312.709,Z 401.53,A -85,B 0,C 180,E1 -15744.838,E2 -15744.838} C_VEL
LIN {X 0,Y 312.982,Z 401.497,A -85,B 0,C 180,E1 -15748.709,E2 -15748.709} C_VEL
LIN {X 0,Y 312.983,Z 401.495,A -85,B 0,C 180,E1 -15751.282,E2 -15751.282} C_VEL
LIN {X 0,Y 312.708,Z 401.53,A -85,B 0,C 180,E1 -15755.153,E2 -15755.153} C_VEL
LIN {X 0,Y 312.861,Z 401.513,A -85,B 0,C 180,E1 -15757.741,E2 -15757.741} C_VEL
LIN {X 0,Y 312.66,Z 401.538,A -85,B 0,C 180,E1 -15761.666,E2 -15761.666} C_VEL
LIN {X 0,Y 312.686,Z 401.532,A -85,B 0,C 180,E1 -15764.883,E2 -15764.883} C_VEL
LIN {X 0,Y 312.614,Z 401.541,A -85,B 0,C 180,E1 -15769.232,E2 -15769.232} C_VEL
LIN {X 0,Y 312.524,Z 401.553,A -85,B 0,C 180,E1 -15772.783,E2 -15772.783} C_VEL
LIN {X 0,Y 312.465,Z 401.565,A -85,B 0,C 180,E1 -15775.887,E2 -15775.887} C_VEL
LIN {X 0,Y 312.203,Z 401.593,A -85,B 0,C 180,E1 -15778.61,E2 -15778.61} C_VEL
LIN {X 0,Y 311.903,Z 401.63,A -85,B 0,C 180,E1 -15781.208,E2 -15781.208} C_VEL
LIN {X 0,Y 311.457,Z 401.925,A -85,B 0,C 180,E1 -15784.334,E2 -15784.334} C_VEL
LIN {X 0,Y 311.352,Z 404.928,A -85,B 0,C 180,E1 -15787.813,E2 -15787.813} C_VEL
LIN {X 0,Y 311.294,Z 407.171,A -85,B 0,C 180,E1 -15790.307,E2 -15790.307} C_VEL
LIN {X 0,Y 314.918,Z 422.419,A -85,B 0,C 180,E1 -15791.299,E2 -15791.299} C_VEL
LIN {X 0,Y 317.565,Z 434.78,A -85,B 0,C 180,E1 -15792.338,E2 -15792.338} C_VEL
LIN {X 0,Y 318.306,Z 439.841,A -85,B 0,C 180,E1 -15792.822,E2 -15792.822} C_VEL
LIN {X 0,Y 317.252,Z 451.058,A -85,B 0,C 180,E1 -15793.95,E2 -15793.95} C_VEL
LIN {X 0,Y 316.015,Z 462.295,A -85,B 0,C 180,E1 -15795.362,E2 -15795.362} C_VEL
LIN {X 0,Y 314.931,Z 472.383,A -85,B 0,C 180,E1 -15796.945,E2 -15796.945} C_VEL
LIN {X 0,Y 313.835,Z 481.248,A -85,B 0,C 180,E1 -15798.655,E2 -15798.655} C_VEL
LIN {X 0,Y 312.826,Z 489.737,A -85,B 0,C 180,E1 -15800.676,E2 -15800.676} C_VEL
LIN {X 0,Y 312.152,Z 496.052,A -85,B 0,C 180,E1 -15802.564,E2 -15802.564} C_VEL
LIN {X 0,Y 311.512,Z 502.245,A -85,B 0,C 180,E1 -15804.948,E2 -15804.948} C_VEL
LIN {X 0,Y 311.142,Z 506.525,A -85,B 0,C 180,E1 -15807.174,E2 -15807.174} C_VEL
LIN {X 0,Y 310.815,Z 509.261,A -85,B 0,C 180,E1 -15809.219,E2 -15809.219} C_VEL
LIN {X 0,Y 310.753,Z 511.117,A -85,B 0,C 180,E1 -15811.646,E2 -15811.646} C_VEL
LIN {X 0,Y 310.763,Z 511.574,A -85,B 0,C 180,E1 -15813.11,E2 -15813.11} C_VEL
LIN {X 0,Y 310.898,Z 511.469,A -85,B 0,C 180,E1 -15814.703,E2 -15814.703} C_VEL
LIN {X 0,Y 311.122,Z 510.927,A -85,B 0,C 180,E1 -15816.01,E2 -15816.01} C_VEL
LIN {X 0,Y 311.515,Z 509.682,A -85,B 0,C 180,E1 -15817.65,E2 -15817.65} C_VEL
LIN {X 0,Y 312.108,Z 507.372,A -85,B 0,C 180,E1 -15819.574,E2 -15819.574} C_VEL
LIN {X 0,Y 312.869,Z 503.736,A -85,B 0,C 180,E1 -15821.672,E2 -15821.672} C_VEL
LIN {X 0,Y 314.191,Z 497.91,A -85,B 0,C 180,E1 -15824.099,E2 -15824.099} C_VEL
LIN {X 0,Y 315.068,Z 493.937,A -85,B 0,C 180,E1 -15825.41,E2 -15825.41} C_VEL
LIN {X 0,Y 315.146,Z 490.95,A -85,B 0,C 180,E1 -15826.335,E2 -15826.335} C_VEL
LIN {X 0,Y 313.641,Z 485.946,A -85,B 0,C 180,E1 -15827.871,E2 -15827.871} C_VEL
LIN {X 0,Y 312.178,Z 480.414,A -85,B 0,C 180,E1 -15829.351,E2 -15829.351} C_VEL
LIN {X 0,Y 312.306,Z 476.58,A -85,B 0,C 180,E1 -15830.175,E2 -15830.175} C_VEL
LIN {X 0,Y 314.224,Z 467.02,A -85,B 0,C 180,E1 -15831.804,E2 -15831.804} C_VEL
LIN {X 0,Y 316.153,Z 456.069,A -85,B 0,C 180,E1 -15833.299,E2 -15833.299} C_VEL
LIN {X 0,Y 317.343,Z 447.516,A -85,B 0,C 180,E1 -15834.282,E2 -15834.282} C_VEL
LIN {X 0,Y 315.041,Z 436.853,A -85,B 0,C 180,E1 -15835.705,E2 -15835.705} C_VEL
LIN {X 0,Y 312.283,Z 428.114,A -85,B 0,C 180,E1 -15836.827,E2 -15836.827} C_VEL
LIN {X 0,Y 306.697,Z 415.392,A -85,B 0,C 180,E1 -15838.483,E2 -15838.483} C_VEL
LIN {X 0,Y 305.613,Z 412.225,A -85,B 0,C 180,E1 -15838.848,E2 -15838.848} C_VEL
LIN {X 0,Y 306.148,Z 410.752,A -85,B 0,C 180,E1 -15841.317,E2 -15841.317} C_VEL
LIN {X 0,Y 306.313,Z 408.09,A -85,B 0,C 180,E1 -15846.589,E2 -15846.589} C_VEL
LIN {X 0,Y 306.376,Z 406.838,A -85,B 0,C 180,E1 -15849.507,E2 -15849.507} C_VEL
LIN {X 0,Y 306.061,Z 405.583,A -85,B 0,C 180,E1 -15853.276,E2 -15853.276} C_VEL
LIN {X 0,Y 305.951,Z 404.874,A -85,B 0,C 180,E1 -15856.002,E2 -15856.002} C_VEL
LIN {X 0,Y 305.869,Z 404.233,A -85,B 0,C 180,E1 -15859.618,E2 -15859.618} C_VEL
LIN {X 0,Y 305.805,Z 404.027,A -85,B 0,C 180,E1 -15863.196,E2 -15863.196} C_VEL
LIN {X 0,Y 305.82,Z 404.191,A -85,B 0,C 180,E1 -15866.345,E2 -15866.345} C_VEL
LIN {X 0,Y 305.879,Z 404.667,A -85,B 0,C 180,E1 -15869.192,E2 -15869.192} C_VEL
LIN {X 0,Y 306.073,Z 405.94,A -85,B 0,C 180,E1 -15873.443,E2 -15873.443} C_VEL
LIN {X 0,Y 306.3,Z 407.362,A -85,B 0,C 180,E1 -15876.625,E2 -15876.625} C_VEL
LIN {X 0,Y 306.686,Z 409.283,A -85,B 0,C 180,E1 -15879.916,E2 -15879.916} C_VEL
LIN {X 0,Y 307.177,Z 411.777,A -85,B 0,C 180,E1 -15883.345,E2 -15883.345} C_VEL
LIN {X 0,Y 307.698,Z 414.936,A -85,B 0,C 180,E1 -15886.963,E2 -15886.963} C_VEL
LIN {X 0,Y 308.286,Z 418.929,A -85,B 0,C 180,E1 -15890.815,E2 -15890.815} C_VEL
LIN {X 0,Y 308.396,Z 422.332,A -85,B 0,C 180,E1 -15893.672,E2 -15893.672} C_VEL
LIN {X 0,Y 307.774,Z 425.446,A -85,B 0,C 180,E1 -15895.989,E2 -15895.989} C_VEL
LIN {X 0,Y 306.66,Z 430.821,A -85,B 0,C 180,E1 -15899.729,E2 -15899.729} C_VEL
LIN {X 0,Y 305.841,Z 436.039,A -85,B 0,C 180,E1 -15903.152,E2 -15903.152} C_VEL
LIN {X 0,Y 306.898,Z 439.813,A -85,B 0,C 180,E1 -15903.492,E2 -15903.492} C_VEL
LIN {X 0,Y 310.61,Z 453.317,A -85,B 0,C 180,E1 -15904.833,E2 -15904.833} C_VEL
LIN {X 0,Y 312.581,Z 464.058,A -85,B 0,C 180,E1 -15905.945,E2 -15905.945} C_VEL
LIN {X 0,Y 313.665,Z 475.555,A -85,B 0,C 180,E1 -15907.233,E2 -15907.233} C_VEL
LIN {X 0,Y 313.614,Z 487.093,A -85,B 0,C 180,E1 -15908.65,E2 -15908.65} C_VEL
LIN {X 0,Y 312.605,Z 494.302,A -85,B 0,C 180,E1 -15909.612,E2 -15909.612} C_VEL
LIN {X 0,Y 310.513,Z 504.615,A -85,B 0,C 180,E1 -15911.19,E2 -15911.19} C_VEL
LIN {X 0,Y 308.719,Z 513.135,A -85,B 0,C 180,E1 -15912.791,E2 -15912.791} C_VEL
LIN {X 0,Y 307.245,Z 521.535,A -85,B 0,C 180,E1 -15914.754,E2 -15914.754} C_VEL
LIN {X 0,Y 305.628,Z 529.491,A -85,B 0,C 180,E1 -15917.049,E2 -15917.049} C_VEL
LIN {X 0,Y 304.583,Z 535.658,A -85,B 0,C 180,E1 -15919.368,E2 -15919.368} C_VEL
LIN {X 0,Y 304.045,Z 539.741,A -85,B 0,C 180,E1 -15921.364,E2 -15921.364} C_VEL
LIN {X 0,Y 303.75,Z 542.804,A -85,B 0,C 180,E1 -15923.362,E2 -15923.362} C_VEL
LIN {X 0,Y 303.687,Z 544.293,A -85,B 0,C 180,E1 -15924.694,E2 -15924.694} C_VEL
LIN {X 0,Y 303.708,Z 545.387,A -85,B 0,C 180,E1 -15926.024,E2 -15926.024} C_VEL
LIN {X 0,Y 303.719,Z 546.082,A -85,B 0,C 180,E1 -15927.352,E2 -15927.352} C_VEL
LIN {X 0,Y 303.819,Z 546.339,A -85,B 0,C 180,E1 -15928.679,E2 -15928.679} C_VEL
LIN {X 0,Y 303.986,Z 546.176,A -85,B 0,C 180,E1 -15930.005,E2 -15930.005} C_VEL
LIN {X 0,Y 303.887,Z 545.593,A -85,B 0,C 180,E1 -15931.33,E2 -15931.33} C_VEL
LIN {X 0,Y 303.773,Z 544.599,A -85,B 0,C 180,E1 -15932.657,E2 -15932.657} C_VEL
LIN {X 0,Y 303.799,Z 543.142,A -85,B 0,C 180,E1 -15933.984,E2 -15933.984} C_VEL
LIN {X 0,Y 303.81,Z 540.292,A -85,B 0,C 180,E1 -15935.886,E2 -15935.886} C_VEL
LIN {X 0,Y 303.98,Z 535.988,A -85,B 0,C 180,E1 -15937.978,E2 -15937.978} C_VEL
LIN {X 0,Y 304.418,Z 529.631,A -85,B 0,C 180,E1 -15940.312,E2 -15940.312} C_VEL
LIN {X 0,Y 305.084,Z 522.691,A -85,B 0,C 180,E1 -15942.308,E2 -15942.308} C_VEL
LIN {X 0,Y 305.875,Z 515.603,A -85,B 0,C 180,E1 -15943.965,E2 -15943.965} C_VEL
LIN {X 0,Y 306.646,Z 508.277,A -85,B 0,C 180,E1 -15945.399,E2 -15945.399} C_VEL
LIN {X 0,Y 308.012,Z 497.745,A -85,B 0,C 180,E1 -15947.088,E2 -15947.088} C_VEL
LIN {X 0,Y 309.307,Z 486.331,A -85,B 0,C 180,E1 -15948.553,E2 -15948.553} C_VEL
LIN {X 0,Y 309.303,Z 480.146,A -85,B 0,C 180,E1 -15949.241,E2 -15949.241} C_VEL
LIN {X 0,Y 308.101,Z 467.011,A -85,B 0,C 180,E1 -15950.488,E2 -15950.488} C_VEL
LIN {X 0,Y 306.492,Z 453.468,A -85,B 0,C 180,E1 -15951.493,E2 -15951.493} C_VEL
LIN {X 0,Y 304.7,Z 440.369,A -85,B 0,C 180,E1 -15952.237,E2 -15952.237} C_VEL
LIN {X 0,Y 305.379,Z 433.781,A -85,B 0,C 180,E1 -15956.16,E2 -15956.16} C_VEL
LIN {X 0,Y 306.286,Z 426.895,A -85,B 0,C 180,E1 -15960.323,E2 -15960.323} C_VEL
LIN {X 0,Y 307.243,Z 421.009,A -85,B 0,C 180,E1 -15963.961,E2 -15963.961} C_VEL
LIN {X 0,Y 307.758,Z 417.132,A -85,B 0,C 180,E1 -15966.427,E2 -15966.427} C_VEL
LIN {X 0,Y 307.412,Z 413.297,A -85,B 0,C 180,E1 -15968.984,E2 -15968.984} C_VEL
LIN {X 0,Y 306.778,Z 409.508,A -85,B 0,C 180,E1 -15971.638,E2 -15971.638} C_VEL
LIN {X 0,Y 305.808,Z 404.339,A -85,B 0,C 180,E1 -15975.438,E2 -15975.438} C_VEL
LIN {X 0,Y 305.493,Z 402.433,A -85,B 0,C 180,E1 -15976.949,E2 -15976.949} C_VEL
LIN {X 0,Y 305.476,Z 402.433,A -85,B 0,C 180,E1 -15981.596,E2 -15981.596} C_VEL
LIN {X 0,Y 305.477,Z 402.433,A -85,B 0,C 180,E1 -15984.888,E2 -15984.888} C_VEL
LIN {X 0,Y 305.458,Z 402.433,A -85,B 0,C 180,E1 -15988.359,E2 -15988.359} C_VEL
LIN {X 0,Y 305.492,Z 402.434,A -85,B 0,C 180,E1 -15991.11,E2 -15991.11} C_VEL
LIN {X 0,Y 305.517,Z 402.425,A -85,B 0,C 180,E1 -15994.082,E2 -15994.082} C_VEL
LIN {X 0,Y 305.491,Z 402.433,A -85,B 0,C 180,E1 -15996.976,E2 -15996.976} C_VEL
LIN {X 0,Y 305.533,Z 402.427,A -85,B 0,C 180,E1 -16001.213,E2 -16001.213} C_VEL
LIN {X 0,Y 305.642,Z 402.412,A -85,B 0,C 180,E1 -16005.348,E2 -16005.348} C_VEL
LIN {X 0,Y 305.64,Z 402.411,A -85,B 0,C 180,E1 -16009.399,E2 -16009.399} C_VEL
LIN {X 0,Y 305.786,Z 402.392,A -85,B 0,C 180,E1 -16012.072,E2 -16012.072} C_VEL
LIN {X 0,Y 305.688,Z 402.408,A -85,B 0,C 180,E1 -16014.722,E2 -16014.722} C_VEL
LIN {X 0,Y 305.966,Z 402.372,A -85,B 0,C 180,E1 -16018.683,E2 -16018.683} C_VEL
LIN {X 0,Y 305.963,Z 402.372,A -85,B 0,C 180,E1 -16021.315,E2 -16021.315} C_VEL
LIN {X 0,Y 305.8,Z 402.393,A -85,B 0,C 180,E1 -16026.597,E2 -16026.597} C_VEL
LIN {X 0,Y 305.708,Z 402.403,A -85,B 0,C 180,E1 -16029.259,E2 -16029.259} C_VEL
LIN {X 0,Y 305.598,Z 402.416,A -85,B 0,C 180,E1 -16033.294,E2 -16033.294} C_VEL
LIN {X 0,Y 305.564,Z 402.42,A -85,B 0,C 180,E1 -16036.02,E2 -16036.02} C_VEL
LIN {X 0,Y 305.495,Z 402.429,A -85,B 0,C 180,E1 -16040.185,E2 -16040.185} C_VEL
LIN {X 0,Y 305.516,Z 402.428,A -85,B 0,C 180,E1 -16044.459,E2 -16044.459} C_VEL
LIN {X 0,Y 305.504,Z 402.428,A -85,B 0,C 180,E1 -16047.392,E2 -16047.392} C_VEL
LIN {X 0,Y 305.447,Z 402.437,A -85,B 0,C 180,E1 -16050.409,E2 -16050.409} C_VEL
LIN {X 0,Y 305.474,Z 402.432,A -85,B 0,C 180,E1 -16054.075,E2 -16054.075} C_VEL
LIN {X 0,Y 305.479,Z 402.434,A -85,B 0,C 180,E1 -16056.737,E2 -16056.737} C_VEL
LIN {X 0,Y 305.462,Z 402.437,A -85,B 0,C 180,E1 -16060.596,E2 -16060.596} C_VEL
LIN {X 0,Y 305.433,Z 402.436,A -85,B 0,C 180,E1 -16063.652,E2 -16063.652} C_VEL
LIN {X 0,Y 305.449,Z 402.434,A -85,B 0,C 180,E1 -16067.413,E2 -16067.413} C_VEL
LIN {X 0,Y 305.464,Z 402.433,A -85,B 0,C 180,E1 -16069.889,E2 -16069.889} C_VEL
LIN {X 0,Y 305.485,Z 402.429,A -85,B 0,C 180,E1 -16073.628,E2 -16073.628} C_VEL
LIN {X 0,Y 305.47,Z 402.436,A -85,B 0,C 180,E1 -16076.479,E2 -16076.479} C_VEL
LIN {X 0,Y 305.461,Z 402.432,A -85,B 0,C 180,E1 -16079.586,E2 -16079.586} C_VEL
LIN {X 0,Y 305.521,Z 402.428,A -85,B 0,C 180,E1 -16082.604,E2 -16082.604} C_VEL
LIN {X 0,Y 305.51,Z 402.426,A -85,B 0,C 180,E1 -16085.534,E2 -16085.534} C_VEL
LIN {X 0,Y 305.519,Z 402.426,A -85,B 0,C 180,E1 -16089.811,E2 -16089.811} C_VEL
LIN {X 0,Y 305.574,Z 402.421,A -85,B 0,C 180,E1 -16092.598,E2 -16092.598} C_VEL
LIN {X 0,Y 305.648,Z 402.409,A -85,B 0,C 180,E1 -16095.344,E2 -16095.344} C_VEL
LIN {X 0,Y 305.633,Z 402.411,A -85,B 0,C 180,E1 -16099.395,E2 -16099.395} C_VEL
LIN {X 0,Y 305.793,Z 402.395,A -85,B 0,C 180,E1 -16102.069,E2 -16102.069} C_VEL
LIN {X 0,Y 305.68,Z 402.406,A -85,B 0,C 180,E1 -16104.719,E2 -16104.719} C_VEL
LIN {X 0,Y 305.949,Z 402.373,A -85,B 0,C 180,E1 -16108.679,E2 -16108.679} C_VEL
LIN {X 0,Y 305.95,Z 402.371,A -85,B 0,C 180,E1 -16111.311,E2 -16111.311} C_VEL
LIN {X 0,Y 305.842,Z 402.386,A -85,B 0,C 180,E1 -16116.593,E2 -16116.593} C_VEL
LIN {X 0,Y 305.725,Z 402.399,A -85,B 0,C 180,E1 -16119.255,E2 -16119.255} C_VEL
LIN {X 0,Y 305.577,Z 402.418,A -85,B 0,C 180,E1 -16123.291,E2 -16123.291} C_VEL
LIN {X 0,Y 305.579,Z 402.423,A -85,B 0,C 180,E1 -16126.015,E2 -16126.015} C_VEL
LIN {X 0,Y 305.56,Z 402.421,A -85,B 0,C 180,E1 -16129.44,E2 -16129.44} C_VEL
LIN {X 0,Y 305.468,Z 402.432,A -85,B 0,C 180,E1 -16133.035,E2 -16133.035} C_VEL
LIN {X 0,Y 305.399,Z 402.444,A -85,B 0,C 180,E1 -16136.173,E2 -16136.173} C_VEL
LIN {X 0,Y 305.11,Z 402.476,A -85,B 0,C 180,E1 -16138.922,E2 -16138.922} C_VEL
LIN {X 0,Y 304.701,Z 402.532,A -85,B 0,C 180,E1 -16142.032,E2 -16142.032} C_VEL
LIN {X 0,Y 304.463,Z 402.562,A -85,B 0,C 180,E1 -16143.801,E2 -16143.801} C_VEL
LIN {X 0,Y 304.339,Z 404.878,A -85,B 0,C 180,E1 -16146.892,E2 -16146.892} C_VEL
LIN {X 0,Y 304.238,Z 407.533,A -85,B 0,C 180,E1 -16149.915,E2 -16149.915} C_VEL
LIN {X 0,Y 308.003,Z 423.314,A -85,B 0,C 180,E1 -16150.989,E2 -16150.989} C_VEL
LIN {X 0,Y 310.611,Z 435.831,A -85,B 0,C 180,E1 -16152.082,E2 -16152.082} C_VEL
LIN {X 0,Y 311.395,Z 439.994,A -85,B 0,C 180,E1 -16152.498,E2 -16152.498} C_VEL
LIN {X 0,Y 310.267,Z 452.126,A -85,B 0,C 180,E1 -16153.755,E2 -16153.755} C_VEL
LIN {X 0,Y 309.011,Z 463.048,A -85,B 0,C 180,E1 -16155.168,E2 -16155.168} C_VEL
LIN {X 0,Y 307.912,Z 473.05,A -85,B 0,C 180,E1 -16156.787,E2 -16156.787} C_VEL
LIN {X 0,Y 306.754,Z 482.213,A -85,B 0,C 180,E1 -16158.608,E2 -16158.608} C_VEL
LIN {X 0,Y 305.863,Z 489.486,A -85,B 0,C 180,E1 -16160.378,E2 -16160.378} C_VEL
LIN {X 0,Y 305.112,Z 496.176,A -85,B 0,C 180,E1 -16162.383,E2 -16162.383} C_VEL
LIN {X 0,Y 304.462,Z 502.293,A -85,B 0,C 180,E1 -16164.756,E2 -16164.756} C_VEL
LIN {X 0,Y 304.058,Z 506.785,A -85,B 0,C 180,E1 -16167.101,E2 -16167.101} C_VEL
LIN {X 0,Y 303.723,Z 509.795,A -85,B 0,C 180,E1 -16169.4,E2 -16169.4} C_VEL
LIN {X 0,Y 303.675,Z 511.453,A -85,B 0,C 180,E1 -16171.561,E2 -16171.561} C_VEL
LIN {X 0,Y 303.73,Z 512.033,A -85,B 0,C 180,E1 -16173.921,E2 -16173.921} C_VEL
LIN {X 0,Y 303.921,Z 511.764,A -85,B 0,C 180,E1 -16175.404,E2 -16175.404} C_VEL
LIN {X 0,Y 304.389,Z 510.557,A -85,B 0,C 180,E1 -16177.434,E2 -16177.434} C_VEL
LIN {X 0,Y 305.132,Z 507.972,A -85,B 0,C 180,E1 -16179.79,E2 -16179.79} C_VEL
LIN {X 0,Y 305.927,Z 504.405,A -85,B 0,C 180,E1 -16181.934,E2 -16181.934} C_VEL
LIN {X 0,Y 307.083,Z 499.577,A -85,B 0,C 180,E1 -16184.061,E2 -16184.061} C_VEL
LIN {X 0,Y 308.571,Z 493.413,A -85,B 0,C 180,E1 -16186.165,E2 -16186.165} C_VEL
LIN {X 0,Y 310.302,Z 485.732,A -85,B 0,C 180,E1 -16188.24,E2 -16188.24} C_VEL
LIN {X 0,Y 312.306,Z 476.58,A -85,B 0,C 180,E1 -16190.175,E2 -16190.175} C_VEL
LIN {X 0,Y 312.477,Z 472.568,A -85,B 0,C 180,E1 -16190.972,E2 -16190.972} C_VEL
LIN {X 0,Y 311.251,Z 465.948,A -85,B 0,C 180,E1 -16192.314,E2 -16192.314} C_VEL
LIN {X 0,Y 310.122,Z 458.952,A -85,B 0,C 180,E1 -16193.574,E2 -16193.574} C_VEL
LIN {X 0,Y 310.412,Z 454.213,A -85,B 0,C 180,E1 -16194.23,E2 -16194.23} C_VEL
LIN {X 0,Y 311.003,Z 449.268,A -85,B 0,C 180,E1 -16194.815,E2 -16194.815} C_VEL
LIN {X 0,Y 308.815,Z 438.815,A -85,B 0,C 180,E1 -16196.289,E2 -16196.289} C_VEL
LIN {X 0,Y 305.972,Z 429.861,A -85,B 0,C 180,E1 -16197.533,E2 -16197.533} C_VEL
LIN {X 0,Y 300.007,Z 416.091,A -85,B 0,C 180,E1 -16199.434,E2 -16199.434} C_VEL
LIN {X 0,Y 298.873,Z 413.252,A -85,B 0,C 180,E1 -16199.79,E2 -16199.79} C_VEL
LIN {X 0,Y 298.81,Z 412.842,A -85,B 0,C 180,E1 -16199.833,E2 -16199.833} C_VEL
LIN {X 0,Y 299.148,Z 411.965,A -85,B 0,C 180,E1 -16201.347,E2 -16201.347} C_VEL
LIN {X 0,Y 299.342,Z 409.357,A -85,B 0,C 180,E1 -16206.743,E2 -16206.743} C_VEL
LIN {X 0,Y 299.404,Z 408.157,A -85,B 0,C 180,E1 -16209.681,E2 -16209.681} C_VEL
LIN {X 0,Y 299.091,Z 406.941,A -85,B 0,C 180,E1 -16213.591,E2 -16213.591} C_VEL
LIN {X 0,Y 298.992,Z 406.285,A -85,B 0,C 180,E1 -16216.385,E2 -16216.385} C_VEL
LIN {X 0,Y 298.921,Z 405.765,A -85,B 0,C 180,E1 -16219.892,E2 -16219.892} C_VEL
LIN {X 0,Y 298.873,Z 405.627,A -85,B 0,C 180,E1 -16223.564,E2 -16223.564} C_VEL
LIN {X 0,Y 298.912,Z 405.878,A -85,B 0,C 180,E1 -16226.704,E2 -16226.704} C_VEL
LIN {X 0,Y 298.973,Z 406.407,A -85,B 0,C 180,E1 -16229.582,E2 -16229.582} C_VEL
LIN {X 0,Y 299.098,Z 407.302,A -85,B 0,C 180,E1 -16232.715,E2 -16232.715} C_VEL
LIN {X 0,Y 299.314,Z 408.682,A -85,B 0,C 180,E1 -16235.946,E2 -16235.946} C_VEL
LIN {X 0,Y 299.694,Z 410.504,A -85,B 0,C 180,E1 -16239.307,E2 -16239.307} C_VEL
LIN {X 0,Y 300.18,Z 412.873,A -85,B 0,C 180,E1 -16242.764,E2 -16242.764} C_VEL
LIN {X 0,Y 300.672,Z 415.936,A -85,B 0,C 180,E1 -16246.437,E2 -16246.437} C_VEL
LIN {X 0,Y 301.242,Z 419.813,A -85,B 0,C 180,E1 -16250.346,E2 -16250.346} C_VEL
LIN {X 0,Y 301.469,Z 422.439,A -85,B 0,C 180,E1 -16252.698,E2 -16252.698} C_VEL
LIN {X 0,Y 301.172,Z 425.024,A -85,B 0,C 180,E1 -16254.761,E2 -16254.761} C_VEL
LIN {X 0,Y 299.795,Z 430.791,A -85,B 0,C 180,E1 -16258.96,E2 -16258.96} C_VEL
LIN {X 0,Y 299.005,Z 435.476,A -85,B 0,C 180,E1 -16262.161,E2 -16262.161} C_VEL
LIN {X 0,Y 300.079,Z 439.187,A -85,B 0,C 180,E1 -16262.516,E2 -16262.516} C_VEL
LIN {X 0,Y 303.583,Z 451.231,A -85,B 0,C 180,E1 -16263.792,E2 -16263.792} C_VEL
LIN {X 0,Y 305.771,Z 461.963,A -85,B 0,C 180,E1 -16264.977,E2 -16264.977} C_VEL
LIN {X 0,Y 307.128,Z 474.542,A -85,B 0,C 180,E1 -16266.431,E2 -16266.431} C_VEL
LIN {X 0,Y 307.179,Z 485.516,A -85,B 0,C 180,E1 -16267.827,E2 -16267.827} C_VEL
LIN {X 0,Y 306.467,Z 492.773,A -85,B 0,C 180,E1 -16268.833,E2 -16268.833} C_VEL
LIN {X 0,Y 304.267,Z 503.218,A -85,B 0,C 180,E1 -16270.438,E2 -16270.438} C_VEL
LIN {X 0,Y 302.306,Z 511.899,A -85,B 0,C 180,E1 -16272.065,E2 -16272.065} C_VEL
LIN {X 0,Y 300.572,Z 520.477,A -85,B 0,C 180,E1 -16274.059,E2 -16274.059} C_VEL
LIN {X 0,Y 299.174,Z 527.46,A -85,B 0,C 180,E1 -16276.073,E2 -16276.073} C_VEL
LIN {X 0,Y 297.819,Z 533.977,A -85,B 0,C 180,E1 -16278.434,E2 -16278.434} C_VEL
LIN {X 0,Y 297.153,Z 538.339,A -85,B 0,C 180,E1 -16280.476,E2 -16280.476} C_VEL
LIN {X 0,Y 296.872,Z 540.68,A -85,B 0,C 180,E1 -16281.839,E2 -16281.839} C_VEL
LIN {X 0,Y 296.624,Z 543.788,A -85,B 0,C 180,E1 -16284.345,E2 -16284.345} C_VEL
LIN {X 0,Y 296.619,Z 545.052,A -85,B 0,C 180,E1 -16285.929,E2 -16285.929} C_VEL
LIN {X 0,Y 296.639,Z 545.696,A -85,B 0,C 180,E1 -16287.289,E2 -16287.289} C_VEL
LIN {X 0,Y 296.726,Z 545.899,A -85,B 0,C 180,E1 -16288.648,E2 -16288.648} C_VEL
LIN {X 0,Y 296.898,Z 545.707,A -85,B 0,C 180,E1 -16290.005,E2 -16290.005} C_VEL
LIN {X 0,Y 296.795,Z 545.093,A -85,B 0,C 180,E1 -16291.362,E2 -16291.362} C_VEL
LIN {X 0,Y 296.693,Z 544.049,A -85,B 0,C 180,E1 -16292.72,E2 -16292.72} C_VEL
LIN {X 0,Y 296.731,Z 542.541,A -85,B 0,C 180,E1 -16294.079,E2 -16294.079} C_VEL
LIN {X 0,Y 296.745,Z 539.873,A -85,B 0,C 180,E1 -16295.886,E2 -16295.886} C_VEL
LIN {X 0,Y 296.926,Z 535.231,A -85,B 0,C 180,E1 -16298.169,E2 -16298.169} C_VEL
LIN {X 0,Y 297.382,Z 528.785,A -85,B 0,C 180,E1 -16300.558,E2 -16300.558} C_VEL
LIN {X 0,Y 298.129,Z 521.719,A -85,B 0,C 180,E1 -16302.6,E2 -16302.6} C_VEL
LIN {X 0,Y 299.167,Z 512.89,A -85,B 0,C 180,E1 -16304.632,E2 -16304.632} C_VEL
LIN {X 0,Y 299.97,Z 504.944,A -85,B 0,C 180,E1 -16306.136,E2 -16306.136} C_VEL
LIN {X 0,Y 301.27,Z 495.181,A -85,B 0,C 180,E1 -16307.658,E2 -16307.658} C_VEL
LIN {X 0,Y 302.505,Z 484.713,A -85,B 0,C 180,E1 -16308.986,E2 -16308.986} C_VEL
LIN {X 0,Y 301.629,Z 472.614,A -85,B 0,C 180,E1 -16310.283,E2 -16310.283} C_VEL
LIN {X 0,Y 300.28,Z 459.788,A -85,B 0,C 180,E1 -16311.391,E2 -16311.391} C_VEL
LIN {X 0,Y 298.539,Z 446.25,A -85,B 0,C 180,E1 -16312.278,E2 -16312.278} C_VEL
LIN {X 0,Y 297.675,Z 440.014,A -85,B 0,C 180,E1 -16312.623,E2 -16312.623} C_VEL
LIN {X 0,Y 298.371,Z 433.542,A -85,B 0,C 180,E1 -16316.59,E2 -16316.59} C_VEL
LIN {X 0,Y 299.212,Z 427.524,A -85,B 0,C 180,E1 -16320.335,E2 -16320.335} C_VEL
LIN {X 0,Y 300.22,Z 421.455,A -85,B 0,C 180,E1 -16324.187,E2 -16324.187} C_VEL
LIN {X 0,Y 300.737,Z 417.806,A -85,B 0,C 180,E1 -16326.557,E2 -16326.557} C_VEL
LIN {X 0,Y 300.298,Z 413.637,A -85,B 0,C 180,E1 -16329.437,E2 -16329.437} C_VEL
LIN {X 0,Y 299.454,Z 408.856,A -85,B 0,C 180,E1 -16332.897,E2 -16332.897} C_VEL
LIN {X 0,Y 298.442,Z 403.36,A -85,B 0,C 180,E1 -16337.117,E2 -16337.117} C_VEL
LIN {X 0,Y 298.401,Z 403.316,A -85,B 0,C 180,E1 -16341.013,E2 -16341.013} C_VEL
LIN {X 0,Y 298.42,Z 403.309,A -85,B 0,C 180,E1 -16343.929,E2 -16343.929} C_VEL
LIN {X 0,Y 298.409,Z 403.316,A -85,B 0,C 180,E1 -16347.2,E2 -16347.2} C_VEL
LIN {X 0,Y 298.419,Z 403.311,A -85,B 0,C 180,E1 -16350.626,E2 -16350.626} C_VEL
LIN {X 0,Y 298.456,Z 403.308,A -85,B 0,C 180,E1 -16354.92,E2 -16354.92} C_VEL
LIN {X 0,Y 298.417,Z 403.31,A -85,B 0,C 180,E1 -16357.862,E2 -16357.862} C_VEL
LIN {X 0,Y 298.48,Z 403.305,A -85,B 0,C 180,E1 -16360.752,E2 -16360.752} C_VEL
LIN {X 0,Y 298.604,Z 403.292,A -85,B 0,C 180,E1 -16364.994,E2 -16364.994} C_VEL
LIN {X 0,Y 298.599,Z 403.29,A -85,B 0,C 180,E1 -16369.146,E2 -16369.146} C_VEL
LIN {X 0,Y 298.732,Z 403.27,A -85,B 0,C 180,E1 -16371.884,E2 -16371.884} C_VEL
LIN {X 0,Y 298.657,Z 403.282,A -85,B 0,C 180,E1 -16374.598,E2 -16374.598} C_VEL
LIN {X 0,Y 298.933,Z 403.248,A -85,B 0,C 180,E1 -16378.652,E2 -16378.652} C_VEL
LIN {X 0,Y 298.93,Z 403.248,A -85,B 0,C 180,E1 -16381.346,E2 -16381.346} C_VEL
LIN {X 0,Y 298.749,Z 403.273,A -85,B 0,C 180,E1 -16386.754,E2 -16386.754} C_VEL
LIN {X 0,Y 298.639,Z 403.283,A -85,B 0,C 180,E1 -16389.48,E2 -16389.48} C_VEL
LIN {X 0,Y 298.557,Z 403.292,A -85,B 0,C 180,E1 -16393.614,E2 -16393.614} C_VEL
LIN {X 0,Y 298.497,Z 403.302,A -85,B 0,C 180,E1 -16396.41,E2 -16396.41} C_VEL
LIN {X 0,Y 298.458,Z 403.305,A -85,B 0,C 180,E1 -16399.616,E2 -16399.616} C_VEL
LIN {X 0,Y 298.441,Z 403.306,A -85,B 0,C 180,E1 -16403.598,E2 -16403.598} C_VEL
LIN {X 0,Y 298.495,Z 403.304,A -85,B 0,C 180,E1 -16406.572,E2 -16406.572} C_VEL
LIN {X 0,Y 298.415,Z 403.31,A -85,B 0,C 180,E1 -16409.64,E2 -16409.64} C_VEL
LIN {X 0,Y 298.403,Z 403.315,A -85,B 0,C 180,E1 -16412.798,E2 -16412.798} C_VEL
LIN {X 0,Y 298.451,Z 403.309,A -85,B 0,C 180,E1 -16416.803,E2 -16416.803} C_VEL
LIN {X 0,Y 298.394,Z 403.314,A -85,B 0,C 180,E1 -16421.084,E2 -16421.084} C_VEL
LIN {X 0,Y 298.407,Z 403.312,A -85,B 0,C 180,E1 -16423.1,E2 -16423.1} C_VEL
LIN {X 0,Y 298.381,Z 403.316,A -85,B 0,C 180,E1 -16426.912,E2 -16426.912} C_VEL
LIN {X 0,Y 298.404,Z 403.313,A -85,B 0,C 180,E1 -16431.004,E2 -16431.004} C_VEL
LIN {X 0,Y 298.423,Z 403.31,A -85,B 0,C 180,E1 -16433.926,E2 -16433.926} C_VEL
LIN {X 0,Y 298.398,Z 403.313,A -85,B 0,C 180,E1 -16437.98,E2 -16437.98} C_VEL
LIN {X 0,Y 298.462,Z 403.306,A -85,B 0,C 180,E1 -16441.9,E2 -16441.9} C_VEL
LIN {X 0,Y 298.488,Z 403.301,A -85,B 0,C 180,E1 -16444.92,E2 -16444.92} C_VEL
LIN {X 0,Y 298.459,Z 403.305,A -85,B 0,C 180,E1 -16449.311,E2 -16449.311} C_VEL
LIN {X 0,Y 298.537,Z 403.299,A -85,B 0,C 180,E1 -16452.175,E2 -16452.175} C_VEL
LIN {X 0,Y 298.592,Z 403.288,A -85,B 0,C 180,E1 -16454.99,E2 -16454.99} C_VEL
LIN {X 0,Y 298.589,Z 403.288,A -85,B 0,C 180,E1 -16459.142,E2 -16459.142} C_VEL
LIN {X 0,Y 298.737,Z 403.272,A -85,B 0,C 180,E1 -16461.881,E2 -16461.881} C_VEL
LIN {X 0,Y 298.651,Z 403.283,A -85,B 0,C 180,E1 -16464.594,E2 -16464.594} C_VEL
LIN {X 0,Y 298.915,Z 403.249,A -85,B 0,C 180,E1 -16468.648,E2 -16468.648} C_VEL
LIN {X 0,Y 298.916,Z 403.247,A -85,B 0,C 180,E1 -16471.342,E2 -16471.342} C_VEL
LIN {X 0,Y 298.788,Z 403.264,A -85,B 0,C 180,E1 -16476.749,E2 -16476.749} C_VEL
LIN {X 0,Y 298.669,Z 403.279,A -85,B 0,C 180,E1 -16479.475,E2 -16479.475} C_VEL
